	// PMC Warnings St.1
	_CheckFanucPMCActiveAlarmList_St01_Wrn : FB_CheckFanucPMCActiveEvents (
						CheckInterval := T#0S, 
						CurrentPMCActiveAlarmList := _CurrentPMCActiveAlarmListCopy,
						PreviousPMCActiveAlarmList := _PreviousPMCActiveAlarmList,
						StartByte := 410,
						ByteLength := 2,
						SourceId := 101,
						SourceName := 'PMC',
						EventClass := ADR(TC_Events.Wrn01),
						EventDetailer := THIS^
						);
	
	// PMC Warnings St.2
	_CheckFanucPMCActiveAlarmList_St02_Wrn : FB_CheckFanucPMCActiveEvents (
						CheckInterval := T#0S, 
						CurrentPMCActiveAlarmList := _CurrentPMCActiveAlarmListCopy,
						PreviousPMCActiveAlarmList := _PreviousPMCActiveAlarmList,
						StartByte := 412,
						ByteLength := 2,
						SourceId := 102,
						SourceName := 'PMC',
						EventClass := ADR(TC_Events.Wrn02),
						EventDetailer := THIS^
						);
	
	// PMC Warnings St.3
	_CheckFanucPMCActiveAlarmList_St03_Wrn : FB_CheckFanucPMCActiveEvents (
						CheckInterval := T#0S, 
						CurrentPMCActiveAlarmList := _CurrentPMCActiveAlarmListCopy,
						PreviousPMCActiveAlarmList := _PreviousPMCActiveAlarmList,
						StartByte := 414,
						ByteLength := 2,
						SourceId := 103,
						SourceName := 'PMC',
						EventClass := ADR(TC_Events.Wrn03),
						EventDetailer := THIS^
						);
	
	// PMC Warnings St.4
	_CheckFanucPMCActiveAlarmList_St04_Wrn : FB_CheckFanucPMCActiveEvents (
						CheckInterval := T#0S, 
						CurrentPMCActiveAlarmList := _CurrentPMCActiveAlarmListCopy,
						PreviousPMCActiveAlarmList := _PreviousPMCActiveAlarmList,
						StartByte := 416,
						ByteLength := 2,
						SourceId := 104,
						SourceName := 'PMC',
						EventClass := ADR(TC_Events.Wrn04),
						EventDetailer := THIS^
						);
	
	// PMC Warnings St.5
	_CheckFanucPMCActiveAlarmList_St05_Wrn : FB_CheckFanucPMCActiveEvents (
						CheckInterval := T#0S, 
						CurrentPMCActiveAlarmList := _CurrentPMCActiveAlarmListCopy,
						PreviousPMCActiveAlarmList := _PreviousPMCActiveAlarmList,
						StartByte := 418,
						ByteLength := 2,
						SourceId := 105,
						SourceName := 'PMC',
						EventClass := ADR(TC_Events.Wrn05),
						EventDetailer := THIS^
						);
	
	// PMC Warnings St.6
	_CheckFanucPMCActiveAlarmList_St06_Wrn : FB_CheckFanucPMCActiveEvents (
						CheckInterval := T#0S, 
						CurrentPMCActiveAlarmList := _CurrentPMCActiveAlarmListCopy,
						PreviousPMCActiveAlarmList := _PreviousPMCActiveAlarmList,
						StartByte := 420,
						ByteLength := 2,
						SourceId := 106,
						SourceName := 'PMC',
						EventClass := ADR(TC_Events.Wrn06),
						EventDetailer := THIS^
						);
	
	// PMC Warnings St.7
	_CheckFanucPMCActiveAlarmList_St07_Wrn : FB_CheckFanucPMCActiveEvents (
						CheckInterval := T#0S, 
						CurrentPMCActiveAlarmList := _CurrentPMCActiveAlarmListCopy,
						PreviousPMCActiveAlarmList := _PreviousPMCActiveAlarmList,
						StartByte := 422,
						ByteLength := 2,
						SourceId := 107,
						SourceName := 'PMC',
						EventClass := ADR(TC_Events.Wrn07),
						EventDetailer := THIS^
						);
	
	// PMC Warnings St.8
	_CheckFanucPMCActiveAlarmList_St08_Wrn : FB_CheckFanucPMCActiveEvents (
						CheckInterval := T#0S, 
						CurrentPMCActiveAlarmList := _CurrentPMCActiveAlarmListCopy,
						PreviousPMCActiveAlarmList := _PreviousPMCActiveAlarmList,
						StartByte := 424,
						ByteLength := 2,
						SourceId := 108,
						SourceName := 'PMC',
						EventClass := ADR(TC_Events.Wrn08),
						EventDetailer := THIS^
						);
	
	// PMC Warnings St.9
	_CheckFanucPMCActiveAlarmList_St09_Wrn : FB_CheckFanucPMCActiveEvents (
						CheckInterval := T#0S, 
						CurrentPMCActiveAlarmList := _CurrentPMCActiveAlarmListCopy,
						PreviousPMCActiveAlarmList := _PreviousPMCActiveAlarmList,
						StartByte := 426,
						ByteLength := 2,
						SourceId := 109,
						SourceName := 'PMC',
						EventClass := ADR(TC_Events.Wrn09),
						EventDetailer := THIS^
						);
	
	// PMC Warnings St.10
	_CheckFanucPMCActiveAlarmList_St10_Wrn : FB_CheckFanucPMCActiveEvents (
						CheckInterval := T#0S, 
						CurrentPMCActiveAlarmList := _CurrentPMCActiveAlarmListCopy,
						PreviousPMCActiveAlarmList := _PreviousPMCActiveAlarmList,
						StartByte := 428,
						ByteLength := 2,
						SourceId := 110,
						SourceName := 'PMC',
						EventClass := ADR(TC_Events.Wrn10),
						EventDetailer := THIS^
						);
	
	// PMC Warnings St.11
	_CheckFanucPMCActiveAlarmList_St11_Wrn : FB_CheckFanucPMCActiveEvents (
						CheckInterval := T#0S, 
						CurrentPMCActiveAlarmList := _CurrentPMCActiveAlarmListCopy,
						PreviousPMCActiveAlarmList := _PreviousPMCActiveAlarmList,
						StartByte := 430,
						ByteLength := 2,
						SourceId := 111,
						SourceName := 'PMC',
						EventClass := ADR(TC_Events.Wrn11),
						EventDetailer := THIS^
						);
	
	// PMC Warnings St.12
	_CheckFanucPMCActiveAlarmList_St12_Wrn : FB_CheckFanucPMCActiveEvents (
						CheckInterval := T#0S, 
						CurrentPMCActiveAlarmList := _CurrentPMCActiveAlarmListCopy,
						PreviousPMCActiveAlarmList := _PreviousPMCActiveAlarmList,
						StartByte := 432,
						ByteLength := 2,
						SourceId := 112,
						SourceName := 'PMC',
						EventClass := ADR(TC_Events.Wrn12),
						EventDetailer := THIS^
						);
	
	// PMC Warnings St.13
	_CheckFanucPMCActiveAlarmList_St13_Wrn : FB_CheckFanucPMCActiveEvents (
						CheckInterval := T#0S, 
						CurrentPMCActiveAlarmList := _CurrentPMCActiveAlarmListCopy,
						PreviousPMCActiveAlarmList := _PreviousPMCActiveAlarmList,
						StartByte := 434,
						ByteLength := 2,
						SourceId := 113,
						SourceName := 'PMC',
						EventClass := ADR(TC_Events.Wrn13),
						EventDetailer := THIS^
						);
	
//	// PMC Warnings St.14
//	_CheckFanucPMCActiveAlarmList_St14_Wrn : FB_CheckFanucPMCActiveEvents (
//						CheckInterval := T#0S, 
//						CurrentPMCActiveAlarmList := _CurrentPMCActiveAlarmListCopy,
//						PreviousPMCActiveAlarmList := _PreviousPMCActiveAlarmList,
//						StartByte := 436,
//						ByteLength := 2,
//						SourceId := 114,
//						SourceName := 'PMC',
//						EventClass := ADR(TC_Events.Wrn14),
//						EventDetailer := THIS^
//						);
	
//	// PMC Warnings St.15
//	_CheckFanucPMCActiveAlarmList_St15_Wrn : FB_CheckFanucPMCActiveEvents (
//						CheckInterval := T#0S, 
//						CurrentPMCActiveAlarmList := _CurrentPMCActiveAlarmListCopy,
//						PreviousPMCActiveAlarmList := _PreviousPMCActiveAlarmList,
//						StartByte := 438,
//						ByteLength := 2,
//						SourceId := 115,
//						SourceName := 'PMC',
//						EventClass := ADR(TC_Events.Wrn15),
//						EventDetailer := THIS^
//						);
	
//	// PMC Warnings St.16
//	_CheckFanucPMCActiveAlarmList_St16_Wrn : FB_CheckFanucPMCActiveEvents (
//						CheckInterval := T#0S, 
//						CurrentPMCActiveAlarmList := _CurrentPMCActiveAlarmListCopy,
//						PreviousPMCActiveAlarmList := _PreviousPMCActiveAlarmList,
//						StartByte := 440,
//						ByteLength := 2,
//						SourceId := 116,
//						SourceName := 'PMC',
//						EventClass := ADR(TC_Events.Wrn16),
//						EventDetailer := THIS^
//						);
	
//	// PMC Warnings St.17
//	_CheckFanucPMCActiveAlarmList_St17_Wrn : FB_CheckFanucPMCActiveEvents (
//						CheckInterval := T#0S, 
//						CurrentPMCActiveAlarmList := _CurrentPMCActiveAlarmListCopy,
//						PreviousPMCActiveAlarmList := _PreviousPMCActiveAlarmList,
//						StartByte := 442,
//						ByteLength := 2,
//						SourceId := 117,
//						SourceName := 'PMC',
//						EventClass := ADR(TC_Events.Wrn17),
//						EventDetailer := THIS^
//						);
	
//	// PMC Warnings St.18
//	_CheckFanucPMCActiveAlarmList_St18_Wrn : FB_CheckFanucPMCActiveEvents (
//						CheckInterval := T#0S, 
//						CurrentPMCActiveAlarmList := _CurrentPMCActiveAlarmListCopy,
//						PreviousPMCActiveAlarmList := _PreviousPMCActiveAlarmList,
//						StartByte := 444,
//						ByteLength := 2,
//						SourceId := 118,
//						SourceName := 'PMC',
//						EventClass := ADR(TC_Events.Wrn18),
//						EventDetailer := THIS^
//						);
	
//	// PMC Warnings St.19
//	_CheckFanucPMCActiveAlarmList_St19_Wrn : FB_CheckFanucPMCActiveEvents (
//						CheckInterval := T#0S, 
//						CurrentPMCActiveAlarmList := v,
//						PreviousPMCActiveAlarmList := _PreviousPMCActiveAlarmList,
//						StartByte := 446,
//						ByteLength := 2,
//						SourceId := 119,
//						SourceName := 'PMC',
//						EventClass := ADR(TC_Events.Wrn19),
//						EventDetailer := THIS^
//						);
	

						
	// TODO: comment out
	_Gen_Alr  AT %MB600:  ARRAY [0..59] OF BYTE;
	_St00_Alr AT %MB660:  ARRAY [0..39] OF BYTE;
	_St01_Alr AT %MB700:  ARRAY [0..9] OF BYTE;
	_St02_Alr AT %MB710:  ARRAY [0..9] OF BYTE;
	_St03_Alr AT %MB720:  ARRAY [0..9] OF BYTE;
	_St04_Alr AT %MB730:  ARRAY [0..9] OF BYTE;
	_St05_Alr AT %MB740:  ARRAY [0..9] OF BYTE;
	_St06_Alr AT %MB750:  ARRAY [0..9] OF BYTE;
	_St07_Alr AT %MB760:  ARRAY [0..9] OF BYTE;
	_St08_Alr AT %MB770:  ARRAY [0..9] OF BYTE;
	_St09_Alr AT %MB780:  ARRAY [0..9] OF BYTE;
	_St10_Alr AT %MB790:  ARRAY [0..9] OF BYTE;
	_St11_Alr AT %MB800:  ARRAY [0..9] OF BYTE;
	_St12_Alr AT %MB810:  ARRAY [0..9] OF BYTE;
	_St13_Alr AT %MB820:  ARRAY [0..9] OF BYTE;
//	_St14_Alr AT %MB830:  ARRAY [0..9] OF BYTE;
//	_St15_Alr AT %MB840:  ARRAY [0..9] OF BYTE;
//	_St16_Alr AT %MB850:  ARRAY [0..9] OF BYTE;
//	_St17_Alr AT %MB860:  ARRAY [0..9] OF BYTE;
//	_St18_Alr AT %MB870:  ARRAY [0..9] OF BYTE;
//	_St19_Alr AT %MB880:  ARRAY [0..9] OF BYTE;
                         
	_Gen_Wrn  AT %MB1000: ARRAY [0..9] OF BYTE;
	_St01_Wrn AT %MB1010: ARRAY [0..1] OF BYTE;
	_St02_Wrn AT %MB1012: ARRAY [0..1] OF BYTE;
	_St03_Wrn AT %MB1014: ARRAY [0..1] OF BYTE;
	_St04_Wrn AT %MB1016: ARRAY [0..1] OF BYTE;
	_St05_Wrn AT %MB1018: ARRAY [0..1] OF BYTE;
	_St06_Wrn AT %MB1020: ARRAY [0..1] OF BYTE;
	_St07_Wrn AT %MB1022: ARRAY [0..1] OF BYTE;
	_St08_Wrn AT %MB1024: ARRAY [0..1] OF BYTE;
	_St09_Wrn AT %MB1026: ARRAY [0..1] OF BYTE;
	_St10_Wrn AT %MB1028: ARRAY [0..1] OF BYTE;
	_St11_Wrn AT %MB1030: ARRAY [0..1] OF BYTE;
	_St12_Wrn AT %MB1032: ARRAY [0..1] OF BYTE;
	_St13_Wrn AT %MB1034: ARRAY [0..1] OF BYTE;
//	_St14_Wrn AT %MB1036: ARRAY [0..1] OF BYTE;
//	_St15_Wrn AT %MB1038: ARRAY [0..1] OF BYTE;
//	_St16_Wrn AT %MB1040: ARRAY [0..1] OF BYTE;
//	_St17_Wrn AT %MB1042: ARRAY [0..1] OF BYTE;
//	_St18_Wrn AT %MB1044: ARRAY [0..1] OF BYTE;
//	_St19_Wrn AT %MB1046: ARRAY [0..1] OF BYTE;

END_VAR

_CheckTimer();

IF Enabled  AND (_CheckInterval > T#0MS) THEN
	IF _CheckTimer.Q THEN
		// Freeze current list into local copy to avoid concurrency problems with ADS
		MEMCPY(ADR(_CurrentPMCActiveAlarmListCopy), ADR(_CurrentPMCActiveAlarmList), NUM_PMC_EVENTS / 8);
		// Update all
		UpdateActiveEventList();
		_CheckTimer.IN := FALSE;
	ELSE
		_CheckTimer.IN := TRUE;
	END_IF
ELSE
	_CheckTimer.IN := FALSE;
END_IF


// Alarms (cyclic call)
_CheckFanucPMCActiveAlarmList_Gen_Alr();
_CheckFanucPMCActiveAlarmList_St00_Alr();
_CheckFanucPMCActiveAlarmList_St01_Alr();
_CheckFanucPMCActiveAlarmList_St02_Alr();
_CheckFanucPMCActiveAlarmList_St03_Alr();
_CheckFanucPMCActiveAlarmList_St04_Alr();
_CheckFanucPMCActiveAlarmList_St05_Alr();
_CheckFanucPMCActiveAlarmList_St06_Alr();
_CheckFanucPMCActiveAlarmList_St07_Alr();
_CheckFanucPMCActiveAlarmList_St08_Alr();
_CheckFanucPMCActiveAlarmList_St09_Alr();
_CheckFanucPMCActiveAlarmList_St10_Alr();
_CheckFanucPMCActiveAlarmList_St11_Alr();
_CheckFanucPMCActiveAlarmList_St12_Alr();
_CheckFanucPMCActiveAlarmList_St13_Alr();
//_CheckFanucPMCActiveAlarmList_St14_Alr();
//_CheckFanucPMCActiveAlarmList_St15_Alr();
//_CheckFanucPMCActiveAlarmList_St16_Alr();
//_CheckFanucPMCActiveAlarmList_St17_Alr();
//_CheckFanucPMCActiveAlarmList_St18_Alr();
//_CheckFanucPMCActiveAlarmList_St19_Alr();

// Warnings (cyclic call)
_CheckFanucPMCActiveAlarmList_Gen_Wrn();
_CheckFanucPMCActiveAlarmList_St01_Wrn();
_CheckFanucPMCActiveAlarmList_St02_Wrn();
_CheckFanucPMCActiveAlarmList_St03_Wrn();
_CheckFanucPMCActiveAlarmList_St04_Wrn();
_CheckFanucPMCActiveAlarmList_St05_Wrn();
_CheckFanucPMCActiveAlarmList_St06_Wrn();
_CheckFanucPMCActiveAlarmList_St07_Wrn();
_CheckFanucPMCActiveAlarmList_St08_Wrn();
_CheckFanucPMCActiveAlarmList_St09_Wrn();
_CheckFanucPMCActiveAlarmList_St10_Wrn();
_CheckFanucPMCActiveAlarmList_St11_Wrn();
_CheckFanucPMCActiveAlarmList_St12_Wrn();
_CheckFanucPMCActiveAlarmList_St13_Wrn();
//_CheckFanucPMCActiveAlarmList_St14_Wrn();
//_CheckFanucPMCActiveAlarmList_St15_Wrn();
//_CheckFanucPMCActiveAlarmList_St16_Wrn();
//_CheckFanucPMCActiveAlarmList_St17_Wrn();
//_CheckFanucPMCActiveAlarmList_St18_Wrn();
//_CheckFanucPMCActiveAlarmList_St19_Wrn();

PROPERTY PUBLIC CheckInterval : TIME
GET
CheckInterval := _CheckInterval;
END_GET
SET
_CheckTimer.PT := _CheckInterval;

//// Alarms
//_CheckFanucPMCActiveAlarmList_Gen_Alr.CheckInterval := _CheckInterval;
//_CheckFanucPMCActiveAlarmList_St00_Alr.CheckInterval := _CheckInterval;
//_CheckFanucPMCActiveAlarmList_St01_Alr.CheckInterval := _CheckInterval;
//_CheckFanucPMCActiveAlarmList_St02_Alr.CheckInterval := _CheckInterval;
//_CheckFanucPMCActiveAlarmList_St03_Alr.CheckInterval := _CheckInterval;
//_CheckFanucPMCActiveAlarmList_St04_Alr.CheckInterval := _CheckInterval;
//_CheckFanucPMCActiveAlarmList_St05_Alr.CheckInterval := _CheckInterval;
//_CheckFanucPMCActiveAlarmList_St06_Alr.CheckInterval := _CheckInterval;
//_CheckFanucPMCActiveAlarmList_St07_Alr.CheckInterval := _CheckInterval;
//_CheckFanucPMCActiveAlarmList_St08_Alr.CheckInterval := _CheckInterval;
//_CheckFanucPMCActiveAlarmList_St09_Alr.CheckInterval := _CheckInterval;
//_CheckFanucPMCActiveAlarmList_St10_Alr.CheckInterval := _CheckInterval;
//_CheckFanucPMCActiveAlarmList_St11_Alr.CheckInterval := _CheckInterval;
//_CheckFanucPMCActiveAlarmList_St12_Alr.CheckInterval := _CheckInterval;
//_CheckFanucPMCActiveAlarmList_St13_Alr.CheckInterval := _CheckInterval;
//_CheckFanucPMCActiveAlarmList_St14_Alr.CheckInterval := _CheckInterval;
//_CheckFanucPMCActiveAlarmList_St15_Alr.CheckInterval := _CheckInterval;
//_CheckFanucPMCActiveAlarmList_St16_Alr.CheckInterval := _CheckInterval;
////_CheckFanucPMCActiveAlarmList_St17_Alr.CheckInterval := _CheckInterval;
////_CheckFanucPMCActiveAlarmList_St18_Alr.CheckInterval := _CheckInterval;
////_CheckFanucPMCActiveAlarmList_St19_Alr.CheckInterval := _CheckInterval;

//// Warnings
//_CheckFanucPMCActiveAlarmList_Gen_Wrn.CheckInterval := _CheckInterval;
//_CheckFanucPMCActiveAlarmList_St01_Wrn.CheckInterval := _CheckInterval;
//_CheckFanucPMCActiveAlarmList_St02_Wrn.CheckInterval := _CheckInterval;
//_CheckFanucPMCActiveAlarmList_St03_Wrn.CheckInterval := _CheckInterval;
//_CheckFanucPMCActiveAlarmList_St04_Wrn.CheckInterval := _CheckInterval;
//_CheckFanucPMCActiveAlarmList_St05_Wrn.CheckInterval := _CheckInterval;
//_CheckFanucPMCActiveAlarmList_St06_Wrn.CheckInterval := _CheckInterval;
//_CheckFanucPMCActiveAlarmList_St07_Wrn.CheckInterval := _CheckInterval;
//_CheckFanucPMCActiveAlarmList_St08_Wrn.CheckInterval := _CheckInterval;
//_CheckFanucPMCActiveAlarmList_St09_Wrn.CheckInterval := _CheckInterval;
//_CheckFanucPMCActiveAlarmList_St10_Wrn.CheckInterval := _CheckInterval;
//_CheckFanucPMCActiveAlarmList_St11_Wrn.CheckInterval := _CheckInterval;
//_CheckFanucPMCActiveAlarmList_St12_Wrn.CheckInterval := _CheckInterval;
//_CheckFanucPMCActiveAlarmList_St13_Wrn.CheckInterval := _CheckInterval;
//_CheckFanucPMCActiveAlarmList_St14_Wrn.CheckInterval := _CheckInterval;
//_CheckFanucPMCActiveAlarmList_St15_Wrn.CheckInterval := _CheckInterval;
//_CheckFanucPMCActiveAlarmList_St16_Wrn.CheckInterval := _CheckInterval;
////_CheckFanucPMCActiveAlarmList_St17_Wrn.CheckInterval := _CheckInterval;
////_CheckFanucPMCActiveAlarmList_St18_Wrn.CheckInterval := _CheckInterval;
////_CheckFanucPMCActiveAlarmList_St19_Wrn.CheckInterval := _CheckInterval;
END_SET
END_PROPERTY

METHOD PUBLIC ClearAll : BOOL
VAR
	_TcEventFilter : FB_TcEventFilter;
END_VAR
// Alarms
_CheckFanucPMCActiveAlarmList_St01_Alr.ClearAll();
_CheckFanucPMCActiveAlarmList_St02_Alr.ClearAll();
_CheckFanucPMCActiveAlarmList_St03_Alr.ClearAll();
_CheckFanucPMCActiveAlarmList_St04_Alr.ClearAll();
_CheckFanucPMCActiveAlarmList_St05_Alr.ClearAll();
_CheckFanucPMCActiveAlarmList_St06_Alr.ClearAll();
_CheckFanucPMCActiveAlarmList_St07_Alr.ClearAll();
_CheckFanucPMCActiveAlarmList_St08_Alr.ClearAll();
_CheckFanucPMCActiveAlarmList_St09_Alr.ClearAll();
_CheckFanucPMCActiveAlarmList_St10_Alr.ClearAll();
_CheckFanucPMCActiveAlarmList_St11_Alr.ClearAll();
_CheckFanucPMCActiveAlarmList_St12_Alr.ClearAll();
_CheckFanucPMCActiveAlarmList_St13_Alr.ClearAll();
//_CheckFanucPMCActiveAlarmList_St14_Alr.ClearAll();
//_CheckFanucPMCActiveAlarmList_St15_Alr.ClearAll();
//_CheckFanucPMCActiveAlarmList_St16_Alr.ClearAll();
//_CheckFanucPMCActiveAlarmList_St17_Alr.ClearAll();
//_CheckFanucPMCActiveAlarmList_St18_Alr.ClearAll();
//_CheckFanucPMCActiveAlarmList_St19_Alr.ClearAll();

// Warnings
_CheckFanucPMCActiveAlarmList_St01_Wrn.ClearAll();
_CheckFanucPMCActiveAlarmList_St02_Wrn.ClearAll();
_CheckFanucPMCActiveAlarmList_St03_Wrn.ClearAll();
_CheckFanucPMCActiveAlarmList_St04_Wrn.ClearAll();
_CheckFanucPMCActiveAlarmList_St05_Wrn.ClearAll();
_CheckFanucPMCActiveAlarmList_St06_Wrn.ClearAll();
_CheckFanucPMCActiveAlarmList_St07_Wrn.ClearAll();
_CheckFanucPMCActiveAlarmList_St08_Wrn.ClearAll();
_CheckFanucPMCActiveAlarmList_St09_Wrn.ClearAll();
_CheckFanucPMCActiveAlarmList_St10_Wrn.ClearAll();
_CheckFanucPMCActiveAlarmList_St11_Wrn.ClearAll();
_CheckFanucPMCActiveAlarmList_St12_Wrn.ClearAll();
_CheckFanucPMCActiveAlarmList_St13_Wrn.ClearAll();
//_CheckFanucPMCActiveAlarmList_St14_Wrn.ClearAll();
//_CheckFanucPMCActiveAlarmList_St15_Wrn.ClearAll();
//_CheckFanucPMCActiveAlarmList_St16_Wrn.ClearAll();
//_CheckFanucPMCActiveAlarmList_St17_Wrn.ClearAll();
//_CheckFanucPMCActiveAlarmList_St18_Wrn.ClearAll();
//_CheckFanucPMCActiveAlarmList_St19_Wrn.ClearAll();
END_METHOD

PROPERTY PUBLIC Enabled : BOOL
GET
Enabled := _Enabled;
END_GET
SET
_Enabled := Enabled;

// Alarms
_CheckFanucPMCActiveAlarmList_Gen_Alr.Enabled := _Enabled;
_CheckFanucPMCActiveAlarmList_St00_Alr.Enabled := _Enabled;
_CheckFanucPMCActiveAlarmList_St01_Alr.Enabled := _Enabled;
_CheckFanucPMCActiveAlarmList_St02_Alr.Enabled := _Enabled;
_CheckFanucPMCActiveAlarmList_St03_Alr.Enabled := _Enabled;
_CheckFanucPMCActiveAlarmList_St04_Alr.Enabled := _Enabled;
_CheckFanucPMCActiveAlarmList_St05_Alr.Enabled := _Enabled;
_CheckFanucPMCActiveAlarmList_St06_Alr.Enabled := _Enabled;
_CheckFanucPMCActiveAlarmList_St07_Alr.Enabled := _Enabled;
_CheckFanucPMCActiveAlarmList_St08_Alr.Enabled := _Enabled;
_CheckFanucPMCActiveAlarmList_St09_Alr.Enabled := _Enabled;
_CheckFanucPMCActiveAlarmList_St10_Alr.Enabled := _Enabled;
_CheckFanucPMCActiveAlarmList_St11_Alr.Enabled := _Enabled;
_CheckFanucPMCActiveAlarmList_St12_Alr.Enabled := _Enabled;
_CheckFanucPMCActiveAlarmList_St13_Alr.Enabled := _Enabled;
//_CheckFanucPMCActiveAlarmList_St14_Alr.Enabled := _Enabled;
//_CheckFanucPMCActiveAlarmList_St15_Alr.Enabled := _Enabled;
//_CheckFanucPMCActiveAlarmList_St16_Alr.Enabled := _Enabled;
//_CheckFanucPMCActiveAlarmList_St17_Alr.Enabled := _Enabled;
//_CheckFanucPMCActiveAlarmList_St18_Alr.Enabled := _Enabled;
//_CheckFanucPMCActiveAlarmList_St19_Alr.Enabled := _Enabled;

// Warnings
_CheckFanucPMCActiveAlarmList_Gen_Wrn.Enabled := _Enabled;
_CheckFanucPMCActiveAlarmList_St01_Wrn.Enabled := _Enabled;
_CheckFanucPMCActiveAlarmList_St02_Wrn.Enabled := _Enabled;
_CheckFanucPMCActiveAlarmList_St03_Wrn.Enabled := _Enabled;
_CheckFanucPMCActiveAlarmList_St04_Wrn.Enabled := _Enabled;
_CheckFanucPMCActiveAlarmList_St05_Wrn.Enabled := _Enabled;
_CheckFanucPMCActiveAlarmList_St06_Wrn.Enabled := _Enabled;
_CheckFanucPMCActiveAlarmList_St07_Wrn.Enabled := _Enabled;
_CheckFanucPMCActiveAlarmList_St08_Wrn.Enabled := _Enabled;
_CheckFanucPMCActiveAlarmList_St09_Wrn.Enabled := _Enabled;
_CheckFanucPMCActiveAlarmList_St10_Wrn.Enabled := _Enabled;
_CheckFanucPMCActiveAlarmList_St11_Wrn.Enabled := _Enabled;
_CheckFanucPMCActiveAlarmList_St12_Wrn.Enabled := _Enabled;
_CheckFanucPMCActiveAlarmList_St13_Wrn.Enabled := _Enabled;
//_CheckFanucPMCActiveAlarmList_St14_Wrn.Enabled := _Enabled;
//_CheckFanucPMCActiveAlarmList_St15_Wrn.Enabled := _Enabled;
//_CheckFanucPMCActiveAlarmList_St16_Wrn.Enabled := _Enabled;
//_CheckFanucPMCActiveAlarmList_St17_Wrn.Enabled := _Enabled;
//_CheckFanucPMCActiveAlarmList_St18_Wrn.Enabled := _Enabled;
//_CheckFanucPMCActiveAlarmList_St19_Wrn.Enabled := _Enabled;
END_SET
END_PROPERTY

METHOD FB_init : BOOL
VAR_INPUT
	bInitRetains : BOOL; // if TRUE, the retain variables are initialized (warm start / cold start)
	bInCopyCode : BOOL;  // if TRUE, the instance afterwards gets moved into the copy code (online change)
	CheckInterval : TIME;
	CurrentPMCActiveAlarmList : REFERENCE TO ARRAY [0..NUM_PMC_EVENTS / 8 - 1] OF BYTE;
END_VAR
_CheckInterval := CheckInterval;
_CheckTimer.PT := _CheckInterval;

IF __ISVALIDREF(CurrentPMCActiveAlarmList) THEN
	_CurrentPMCActiveAlarmList REF= CurrentPMCActiveAlarmList;
END_IF
END_METHOD

METHOD GetDetail : STRING(255)
VAR_INPUT
	TcAlarm	: REFERENCE TO Tc3_EventLogger.FB_TcAlarm;
END_VAR
VAR
	_Detail : STRING(255);
END_VAR
_Detail := '';

// St.01 Alarms
IF TcAlarm.EqualsToEventClass(TC_EVENT_CLASSES.Alr01) THEN
	CASE TcAlarm.nEventId OF
		0: _Detail := 'This is alarm 0 of St.1';
		1: _Detail := 'This is alarm 1 of St.1';
		2: _Detail := 'This is alarm 2 of St.1';
		3: _Detail := 'This is alarm 3 of St.1';
		//4: _Detail := Main._CurrentUser.Name;
		//5: _Detail := GlobalUser.GlobalUser.Name;
	END_CASE
END_IF

// St.01 Warnings
IF TcAlarm.EqualsToEventClass(TC_EVENT_CLASSES.Wrn01) THEN
	CASE TcAlarm.nEventId OF
		0: _Detail := 'This is warning 0 of St.1';
		1: _Detail := 'This is warning 1 of St.1';
		2: _Detail := 'This is warning 2 of St.1';
		3: _Detail := 'This is warning 3 of St.1';
	END_CASE
END_IF

GetDetail := _Detail;
END_METHOD

METHOD PUBLIC ReSync : BOOL
// Force resynchronization of active events
//		- Clear all raised events
//		- Reset previous memory buffer
//		- Update active event list
ClearAll();
MemSet(ADR(_PreviousPMCActiveAlarmList), 0, SIZEOF(_PreviousPMCActiveAlarmList));
UpdateActiveEventList();
END_METHOD

METHOD PUBLIC UpdateActiveEventList : BOOL
// Alarms
_CheckFanucPMCActiveAlarmList_Gen_Alr.UpdateActiveEventList();
_CheckFanucPMCActiveAlarmList_St00_Alr.UpdateActiveEventList();
_CheckFanucPMCActiveAlarmList_St01_Alr.UpdateActiveEventList();
_CheckFanucPMCActiveAlarmList_St02_Alr.UpdateActiveEventList();
_CheckFanucPMCActiveAlarmList_St03_Alr.UpdateActiveEventList();
_CheckFanucPMCActiveAlarmList_St04_Alr.UpdateActiveEventList();
_CheckFanucPMCActiveAlarmList_St05_Alr.UpdateActiveEventList();
_CheckFanucPMCActiveAlarmList_St06_Alr.UpdateActiveEventList();
_CheckFanucPMCActiveAlarmList_St07_Alr.UpdateActiveEventList();
_CheckFanucPMCActiveAlarmList_St08_Alr.UpdateActiveEventList();
_CheckFanucPMCActiveAlarmList_St09_Alr.UpdateActiveEventList();
_CheckFanucPMCActiveAlarmList_St10_Alr.UpdateActiveEventList();
_CheckFanucPMCActiveAlarmList_St11_Alr.UpdateActiveEventList();
_CheckFanucPMCActiveAlarmList_St12_Alr.UpdateActiveEventList();
_CheckFanucPMCActiveAlarmList_St13_Alr.UpdateActiveEventList();
//_CheckFanucPMCActiveAlarmList_St14_Alr.UpdateActiveEventList();
//_CheckFanucPMCActiveAlarmList_St15_Alr.UpdateActiveEventList();
//_CheckFanucPMCActiveAlarmList_St16_Alr.UpdateActiveEventList();
//_CheckFanucPMCActiveAlarmList_St17_Alr.UpdateActiveEventList();
//_CheckFanucPMCActiveAlarmList_St18_Alr.UpdateActiveEventList();
//_CheckFanucPMCActiveAlarmList_St19_Alr.UpdateActiveEventList();

// Warnings
_CheckFanucPMCActiveAlarmList_Gen_Wrn.UpdateActiveEventList();
_CheckFanucPMCActiveAlarmList_St01_Wrn.UpdateActiveEventList();
_CheckFanucPMCActiveAlarmList_St02_Wrn.UpdateActiveEventList();
_CheckFanucPMCActiveAlarmList_St03_Wrn.UpdateActiveEventList();
_CheckFanucPMCActiveAlarmList_St04_Wrn.UpdateActiveEventList();
_CheckFanucPMCActiveAlarmList_St05_Wrn.UpdateActiveEventList();
_CheckFanucPMCActiveAlarmList_St06_Wrn.UpdateActiveEventList();
_CheckFanucPMCActiveAlarmList_St07_Wrn.UpdateActiveEventList();
_CheckFanucPMCActiveAlarmList_St08_Wrn.UpdateActiveEventList();
_CheckFanucPMCActiveAlarmList_St09_Wrn.UpdateActiveEventList();
_CheckFanucPMCActiveAlarmList_St10_Wrn.UpdateActiveEventList();
_CheckFanucPMCActiveAlarmList_St11_Wrn.UpdateActiveEventList();
_CheckFanucPMCActiveAlarmList_St12_Wrn.UpdateActiveEventList();
_CheckFanucPMCActiveAlarmList_St13_Wrn.UpdateActiveEventList();
//_CheckFanucPMCActiveAlarmList_St14_Wrn.UpdateActiveEventList();
//_CheckFanucPMCActiveAlarmList_St15_Wrn.UpdateActiveEventList();
//_CheckFanucPMCActiveAlarmList_St16_Wrn.UpdateActiveEventList();
//_CheckFanucPMCActiveAlarmList_St17_Wrn.UpdateActiveEventList();
//_CheckFanucPMCActiveAlarmList_St18_Wrn.UpdateActiveEventList();
//_CheckFanucPMCActiveAlarmList_St19_Wrn.UpdateActiveEventList();
END_METHOD

END_FUNCTION_BLOCK

// ---- FBs/Events/FB_CheckFanucPMCActiveEvents.TcPOU
FUNCTION_BLOCK FB_CheckFanucPMCActiveEvents
VAR_INPUT
	Enabled : BOOL;
END_VAR
VAR

	{attribute 'hide'}
	_PMCEvents : ARRAY[0..NUM_PMC_EVENTS] OF FB_TcAlarm;

	{attribute 'hide'}
	_CurrentPMCActiveAlarmList : REFERENCE TO ARRAY [0..NUM_PMC_EVENTS / 8 - 1] OF BYTE;

	{attribute 'hide'}
	_PreviousPMCActiveAlarmList : REFERENCE TO ARRAY [0..NUM_PMC_EVENTS / 8 - 1] OF BYTE;
	
	{attribute 'hide'}
	_TcEventLogger : FB_TcEventLogger;	

	{attribute 'hide'}
	_TcSourceInfo : FB_TcSourceInfo;

	{attribute 'hide'}
	_CheckInterval : TIME;
	
	{attribute 'hide'}
	_CheckTimer : TON;
	
	{attribute 'hide'}
	_StartByte : UDINT := 0;

	{attribute 'hide'}
	_ByteLength : UDINT := 0;

	{attribute 'hide'}
	_EventClass : POINTER TO TcEventEntry;
	
	{attribute 'hide'}
	_EventDetailer : I_EventDetailer;
	
END_VAR

_CheckTimer();

IF Enabled  AND (_CheckInterval > T#0MS) THEN
	IF _CheckTimer.Q THEN
		THIS^.UpdateActiveEventList();
		_CheckTimer.IN := FALSE;
	ELSE
		_CheckTimer.IN := TRUE;
	END_IF
ELSE
	_CheckTimer.IN := FALSE;
END_IF

METHOD PRIVATE BinarySearch : BOOL
VAR_INPUT
	FirstByteIndex : UDINT;
	LastByteIndex : UDINT;
END_VAR
VAR 
	_i : UDINT;
	_StateChanged : INT;
	_EventIndex : UDINT;
	_pTcEventEntry : POINTER TO TcEventEntry;
	_MiddleByteIndex : UDINT;
	_TcAlarm : FB_TcAlarm;
	_refTcAlarm : REFERENCE TO FB_TcAlarm REF= _TcAlarm;
	_hr : HRESULT;
END_VAR
IF FirstByteIndex = LastByteIndex THEN
	IF _PreviousPMCActiveAlarmList[FirstByteIndex] <> _CurrentPMCActiveAlarmList[FirstByteIndex] THEN
		// Check every bit for change: (X = 2^BitPos)
		// | Current | Previous | Current - Previous | StateChanged
		// |    0     |    0    |         0          | No change
		// |    0     |    1    |      -X < 0        | Event gone
		// |    1     |    0    |       X > 0        | Event coming
		// |    1     |    1    |         0          | No change
		_pTcEventEntry := _EventClass;
		FOR _i := 0 TO 7 DO
			_StateChanged := BYTE_TO_INT(_CurrentPMCActiveAlarmList[FirstByteIndex] AND SHL(16#1, _i)) - BYTE_TO_INT(_PreviousPMCActiveAlarmList[FirstByteIndex] AND SHL(16#1, _i));
			IF _StateChanged < 0 THEN
				// Event gone
				_EventIndex := (FirstByteIndex - _StartByte) * 8 + _i;
				// Clear event
				IF _PMCEvents[_EventIndex].bRaised THEN
					_PMCEvents[_EventIndex].Clear(0, TRUE);
				END_IF
			END_IF
			IF _StateChanged > 0 THEN
				// Event coming
				_EventIndex := (FirstByteIndex - _StartByte) * 8 + _i;
				// Create event instance if not already created
				IF _PMCEvents[_EventIndex].nUniqueId = 0 THEN
					_PMCEvents[_EventIndex].CreateEx(_pTcEventEntry[_EventIndex], FALSE, GetSourceInfo());
				END_IF
				// Raise event (if not already raised)
				IF NOT _PMCEvents[_EventIndex].bRaised THEN
					SetParameters(_PMCEvents[_EventIndex]);
					_PMCEvents[_EventIndex].Raise(0);
				END_IF
			END_IF		
		END_FOR		
	END_IF
ELSE
	_MiddleByteIndex := FirstByteIndex + LREAL_TO_UDINT(FLOOR((LastByteIndex - FirstByteIndex) / 2));
	// Check first half (recursive)
	IF MEMCMP(ADR(_PreviousPMCActiveAlarmList[FirstByteIndex]), ADR(_CurrentPMCActiveAlarmList[FirstByteIndex]), (_MiddleByteIndex + 1 - FirstByteIndex)) <> 0 THEN
		THIS^.BinarySearch(FirstByteIndex, _MiddleByteIndex);
	END_IF
	// Check second half (recursive)
	IF MEMCMP(ADR(_PreviousPMCActiveAlarmList[_MiddleByteIndex + 1]), ADR(_CurrentPMCActiveAlarmList[_MiddleByteIndex + 1]), (LastByteIndex - _MiddleByteIndex)) <> 0 THEN
		THIS^.BinarySearch(_MiddleByteIndex + 1, LastByteIndex);
	END_IF
END_IF
END_METHOD

PROPERTY PUBLIC ByteLength : UDINT
GET
ByteLength := _ByteLength;
END_GET
END_PROPERTY

PROPERTY PUBLIC CheckInterval : TIME
GET
CheckInterval := _CheckInterval;
END_GET
SET
_CheckInterval := CheckInterval;
_CheckTimer.PT := _CheckInterval;
END_SET
END_PROPERTY

METHOD PUBLIC ClearAll : BOOL
VAR
	_TcEventFilter : FB_TcEventFilter;
END_VAR
//_TcEventFilter.Clear().EventClass.EqualTo(_EventClass);
//_TcEventLogger.ClearAlarms(0, FALSE, _TcEventFilter);
END_METHOD

METHOD FB_init : BOOL
VAR_INPUT
	bInitRetains : BOOL; // if TRUE, the retain variables are initialized (warm start / cold start)
	bInCopyCode : BOOL;  // if TRUE, the instance afterwards gets moved into the copy code (online change)
	CheckInterval : TIME;
	CurrentPMCActiveAlarmList : REFERENCE TO ARRAY [0..NUM_PMC_EVENTS / 8 - 1] OF BYTE;
	PreviousPMCActiveAlarmList : REFERENCE TO ARRAY [0..NUM_PMC_EVENTS / 8 - 1] OF BYTE;
	StartByte : UDINT;
	ByteLength : UDINT;
	SourceId : UDINT := 0;
	SourceName : STRING[80] := '';
	EventClass : POINTER TO TcEventEntry;
	EventDetailer : I_EventDetailer;
END_VAR
_CheckInterval := CheckInterval;
_CheckTimer.PT := _CheckInterval;

_StartByte := StartByte;
_ByteLength := ByteLength;

_EventClass := EventClass;

InitSource(SourceId, SourceName);

IF __ISVALIDREF(CurrentPMCActiveAlarmList) THEN
	_CurrentPMCActiveAlarmList REF= CurrentPMCActiveAlarmList;
END_IF

IF __ISVALIDREF(PreviousPMCActiveAlarmList) THEN
	_PreviousPMCActiveAlarmList REF= PreviousPMCActiveAlarmList;
END_IF

_EventDetailer := EventDetailer;
END_METHOD

METHOD PRIVATE GetSourceInfo : I_TcSourceInfo
GetSourceInfo := _TcSourceInfo;
END_METHOD

METHOD PRIVATE InitSource : BOOL
VAR_INPUT
	Id : UDINT;
	Name : STRING(80);
END_VAR
_TcSourceInfo.Clear();
_TcSourceInfo.nId := ID;
_TcSourceInfo.sName := Name;
END_METHOD

METHOD PRIVATE SetParameters : BOOL
VAR_INPUT
	TcAlarm : REFERENCE TO FB_TcAlarm;
END_VAR
VAR
	_Detail : STRING(512);
END_VAR
IF _EventDetailer <> 0 THEN
	_Detail := _EventDetailer.GetDetail(TcAlarm);
END_IF

TcAlarm.ipArguments.Clear();

IF LEn(_Detail) <> 0 THEN
	TcAlarm.ipArguments.AddString(_Detail);
END_IF
END_METHOD

PROPERTY PUBLIC SourceId : UDINT
GET
SourceId := _TcSourceInfo.nId;
END_GET
END_PROPERTY

PROPERTY PUBLIC SourceName : STRING(80)
GET
SourceName := _TcSourceInfo.sName;
END_GET
END_PROPERTY

PROPERTY PUBLIC StartByte : UDINT
GET
StartByte := _StartByte;
END_GET
END_PROPERTY

METHOD PUBLIC UpdateActiveEventList : BOOL
VAR
	_i : UINT;
	_j : UINT;
	_Found : BOOL;	
	_TcAlarm : FB_TcAlarm;
	_refTcAlarm : REFERENCE TO FB_TcAlarm REF= _TcAlarm;
	_iTcSourceInfo : I_TcSourceInfo;
	_hr : HRESULT;
END_VAR
IF SIZEOF(_PreviousPMCActiveAlarmList) <> SIZEOF(_CurrentPMCActiveAlarmList) THEN
	UpdateActiveEventList := FALSE;
	RETURN;
END_IF

IF MEMCMP(ADR(_PreviousPMCActiveAlarmList) + _StartByte, ADR(_CurrentPMCActiveAlarmList) + _StartByte, _ByteLength) <> 0 THEN
	
	// Explore alarms and manage going and coming
	IF SIZEOF(_CurrentPMCActiveAlarmList) > 0 THEN
		BinarySearch(_StartByte, _StartByte + _ByteLength - 1);
	END_IF
	
	// Update previous list with current list
	MEMCPY(ADR(_PreviousPMCActiveAlarmList) + _StartByte, ADR(_CurrentPMCActiveAlarmList) + _StartByte, _ByteLength);

END_IF

UpdateActiveEventList := TRUE;
END_METHOD

END_FUNCTION_BLOCK

// ---- FBs/Database/PRG_MSSQL_spCMD_AbortProduction.TcPOU
PROGRAM PRG_MSSQL_spCMD_AbortProduction
VAR_INPUT
	Execute					: BOOL;
	Enable					: BOOL;
END_VAR
VAR_OUTPUT
	Error					: BOOL;
	ErrorID					: DINT;
	Done					: BOOL;
	Busy					: BOOL;
	tcMessage 				: I_TcMessage;
	Q_tElapsedTime			: TIME;
END_VAR
VAR
	RTRIG_Execute			: R_TRIG;
	iState					: INT := -1;
	return_value				: DINT;
END_VAR
VAR_IN_OUT
	fbSQLResult				: FB_SQLResultEvt;
	fbSQLStoredProcedure	: FB_SQLStoredProcedureEvt;
END_VAR

RTRIG_Execute(CLK := Execute AND Enable);
IF(RTRIG_Execute.Q) THEN
	 Done							:= FALSE;
	 Error							:= FALSE;
	 ErrorID						:= 0;
	 
	 iState							:= 0;
ELSIF NOT Execute AND NOT Busy THEN
	Busy			:= FALSE;
	Done			:= FALSE;
	Error			:= FALSE;
	
	iState := -1;
END_IF
 
 CASE iState OF
 
	 0:
		Busy								:= TRUE;
		iState 								:= 10;
		
	10:
		IF fbSQLStoredProcedure.ExecuteDataReturn(pParameterStrc := ADR(return_value), cbParameterStrc := SIZEOF(return_value), pSQLDBResult := ADR(fbSqlResult)) THEN
			IF fbSQLStoredProcedure.bError THEN
				tcMessage := fbSQLStoredProcedure.ipTcResult;
				
				iState 							:= 1010;
			ELSE
				iState 							:= 20;
			END_IF    
		END_IF
		
	20:
		IF return_value = 0 THEN
			iState 								:= 999;	
		ELSE
			iState 								:= 1020;	
		END_IF
		
	999:
		Done			:= TRUE;
		Busy			:= FALSE;
		
 END_CASE 
 
IF iState > 1000 THEN
	Error 		:= TRUE;
	ErrorID	 	:= iState;
	Busy	 	:= FALSE;
	iState := -1;
END_IF

END_PROGRAM

// ---- FCs/FC_BYTE_TO_BOOLARR.TcPOU
FUNCTION FC_BYTE_TO_BOOLARR
VAR_INPUT
	pMyBool : POINTER TO BOOL; // Destination 
	pMyByte : POINTER TO BYTE; // Source   
	nSize	: UINT;               
END_VAR
VAR
    i : UINT;                       
	myBools : ARRAY[0..7] OF BOOL; 
END_VAR

FOR i:= 0 TO nSize-1 BY 8 DO
	myBools := FC_BYTE_TO_BOOLBYTE(pMyByte[i/8]);
	MEMCPY(ADR(pMyBool[i]), ADR(myBools), SIZEOF(myBools));
END_FOR

END_FUNCTION

// ---- FCs/FC_BYTE_TO_BOOLBYTE.TcPOU
FUNCTION FC_BYTE_TO_BOOLBYTE : ARRAY[0..7] OF BOOL
VAR_INPUT
	myByte : REFERENCE TO BYTE;
END_VAR
VAR
    i : USINT;
END_VAR

FOR i := 0 TO 7 DO
    FC_BYTE_TO_BOOLBYTE[i] := (myByte AND (SHL(1,i))) <> 0;
END_FOR

END_FUNCTION

// ---- POUs/MAIN_SERVICE.TcPOU
PROGRAM MAIN_SERVICE
VAR
	
// HMI - Tools	
	NT_CNCScreenDisplay: NT_StartProcess;
	NT_ProgramTransferTool: NT_StartProcess;
	NT_TaskManager: NT_StartProcess;
	NT_OnScreenKeyboard: NT_StartProcess;
	NT_CloseBrowser: NT_StartProcess;
	NT_FanucLadder: NT_StartProcess;
	NT_FlyCad: NT_StartProcess;
	NT_OpenExe : NT_StartProcess;
	NT_CloseExe : NT_StartProcess;
	
	TON_OpenPage : TON;
	
	GetTime								: FB_LocalSystemTime := ( bEnable := TRUE, dwCycle := 1 );	
	
	otTON						: OTSTRUCT;
	otTOFF						: OTSTRUCT;
	otTDOWN						: OTSTRUCT;
	otTTotal					: OTSTRUCT;
	TempSum						: REAL;
	TempTime1					: REAL;
	TempTime2					: REAL;
	TempTime3					: REAL;
	RTON_ON					: FB_RetainTimer;
	RTON_OFF				: FB_RetainTimer;
	RTON_DOWN				: FB_RetainTimer;

	fbGetCurTaskIndex : GETCURTASKINDEX;
	
	TON_OvrMultFeedback : TON;
	OvrMultiplierOld	: USINT;
	_iDataPos : INT;
	i : INT;
	RTRIG_ClearAlarm	: R_TRIG;
	TcSourceInfo	: FB_TcSourceInfo;
	fbRefresh : FB_Refresh;
	MSSQL_Events					: DUT_Events;
	Marker_Events					: DUT_Events;
	DataRequest_Events				: DUT_Events;
	
	TON_DelayMarkerConnected	: TON;
	fbDoublingTriggerGood : FB_DoublingTrigger;
	fbDoublingTriggerBad : FB_DoublingTrigger;
	fbHMI_SP_Alarm			: ARRAY[1..DB.MAX_NUMBER_ST] OF FB_HMI_SP_Alarm;
	MSSQL_TcSourceInfo	: ARRAY[1..DB.MAX_NUMBER_ST] OF FB_TcSourceInfo;
	TcEventLogger 	: FB_TcEventLogger;
	RTRIG_BatchChange			: R_TRIG;
END_VAR

fbGetCurTaskIndex();

A_00_Init();
A_10_DiagnosticTools();	// Windows Software tools
A_20_Production();
A_30_SystemTime();
A_92_HMI_Output();
A_99_Alarm();

PRG_EventManagement();

ACTION A_00_Init:
IF _TaskInfo[fbGetCurTaskIndex.index].FirstCycle THEN	// First cycle of this task
	A_99_Alarm_Init();
END_IF
END_ACTION

ACTION A_10_DiagnosticTools:
//UPS Management
PF_00_UPS();

// Launch utility software
NT_CNCScreenDisplay(
	NETID:= '', 
	PATHSTR:= 'C:\Program Files (x86)\CNCScreenE\CNCScrnE.exe', 
	DIRNAME:= '', 
	COMNDLINE:= '', 
	START:= HMI.In.Tools.CNCScreenDisplay, 
	TMOUT:= , 
	BUSY=> HMI.Out.Tools.CNCScreenDisplay, 
	ERR=> , 
	ERRID=> );
	
NT_ProgramTransferTool(
	NETID:= '', 
	PATHSTR:= 'C:\Program Files (x86)\FANUC\Program Transfer Tool\Bin\PttMain.exe', 
	DIRNAME:= '', 
	COMNDLINE:= , 
	START:= HMI.In.Tools.ProgramTransferTool, 
	TMOUT:= , 
	BUSY=> HMI.Out.Tools.ProgramTransferTool, 
	ERR=> , 
	ERRID=> );
	
NT_TaskManager(
	NETID:= , 
	PATHSTR:= 'C:\Windows\system32\Taskmgr.exe', 
	DIRNAME:= '', 
	COMNDLINE:= , 
	START:= HMI.In.Tools.TaskManager, 
	TMOUT:= , 
	BUSY=> HMI.Out.Tools.TaskManager, 
	ERR=> , 
	ERRID=> );
	
NT_OnScreenKeyboard(
	NETID:= , 
	PATHSTR:= 'C:\GSCNext\osk1.bat', 
	DIRNAME:= '', 
	COMNDLINE:= , 
	START:= HMI.In.Tools.OnScreenKeyboard, 
	TMOUT:= , 
	BUSY=> HMI.Out.Tools.OnScreenKeyboard, 
	ERR=> , 
	ERRID=> );
	
NT_CloseBrowser(
	NETID:= , 
	PATHSTR:= 'C:\GSCNext\CloseBrowser.bat', 
	DIRNAME:= '', 
	COMNDLINE:= , 
	START:= HMI.In.Tools.CloseBrowser, 
	TMOUT:= , 
	BUSY=> HMI.Out.Tools.CloseBrowser, 
	ERR=> , 
	ERRID=> );
	
NT_FanucLadder(
	NETID:= , 
	PATHSTR:= 'C:\PROGRAM Files (x86)\FANUC PMC Programmer\FANUC LADDER-3\Fladder.exe', 
	DIRNAME:= '', 
	COMNDLINE:= , 
	START:= HMI.In.Tools.FanucLadder, 
	TMOUT:= , 
	BUSY=> HMI.Out.Tools.FanucLadder, 
	ERR=> , 
	ERRID=> );
	
NT_FlyCad(
	NETID:= , 
	PATHSTR:= 'C:\Program Files (x86)\FlyCAD\flycad.exe', 
	DIRNAME:= '', 
	COMNDLINE:= , 
	START:= HMI.In.Tools.FlyCad, 
	TMOUT:= , 
	BUSY=> HMI.Out.Tools.FlyCad, 
	ERR=> , 
	ERRID=> );

NT_OpenExe( 
	NETID := , 
	PATHSTR := 'C:\GSCNext\UtilityBAT\AperturaExeFromPlc.bat', 
	DIRNAME := 'C:\GSCNext\UtilityBAT', 
	COMNDLINE := , 
	START := , 
	TMOUT := T#5S, 
	BUSY => , 
	ERR => , 
	ERRID =>
);

NT_CloseExe(
	NETID:= , 
	PATHSTR := 'C:\GSCNext\UtilityBAT\ChiusuraExeFromPlc.bat', 
	DIRNAME := 'C:\GSCNext\UtilityBAT', 
	COMNDLINE := , 
	START := , 
	TMOUT := T#5S, 
	BUSY => , 
	ERR => , 
	ERRID => 
);
	
///////////////////////////////////////////////////////////////
TON_OpenPage(IN:= HMI.In.Tools.OpenPage, PT:= T#5S);
HMI.Out.Tools.OpenPage := TON_OpenPage.Q;

///////////////////////////////////////////////////////////////
END_ACTION

ACTION A_20_Production:
fbDoublingTriggerGood(TriggerIn := G.OEE_bCountUpGood);
fbDoublingTriggerBad(TriggerIn := G.OEE_bCountUpBad);

PRG_OEE(Enable := HMI.In.Statistics.OEE_Enable,
		Reset := HMI.In.Statistics.OEE_Reset,
		StartTimer := NOT G.MachineEmpty AND NOT PRG_OEE.Reset,
		bStatusON := HMI.Out.Header.MachineState = eState.Running,
		bStatusOFF := NOT PRG_OEE.bStatusON AND NOT PRG_OEE.bStatusDOWN,
		bStatusDOWN := MachineData.aBool[4],
		tPlannedProductionTime := DWORD_TO_TIME(HMI.Production.OEE.PlannedProductionTime*60000),
		tIdealCycleTime := HMI.Production.OEE.IdealCycleTime,
		bCountUpGood := fbDoublingTriggerGood.TriggerOut,
		bCountUpBad	:= fbDoublingTriggerBad.TriggerOut,
		GoodPieces => HMI.Production.OEE.GoodPieces,
		BadPieces => HMI.Production.OEE.BadPieces,	
);

IF G.OEE_bCountUpGood THEN
	G.OEE_bCountUpGood  := FALSE;
END_IF
IF G.OEE_bCountUpBad THEN
	G.OEE_bCountUpBad  := FALSE;
END_IF

otTON := TIME_TO_OTSTRUCT(PRG_OEE.tON);
otTOFF := TIME_TO_OTSTRUCT(PRG_OEE.tOFF);
otTDOWN := TIME_TO_OTSTRUCT(PRG_OEE.tDOWN);
otTTotal := TIME_TO_OTSTRUCT(PRG_OEE.tON + PRG_OEE.tOFF + PRG_OEE.tDOWN);

HMI.Production.OEE.s_tON 	:= FC_Concat4(WORD_TO_STRING(otTON.wHour) , 'h ',WORD_TO_STRING(otTON.wMinute), 'm');
HMI.Production.OEE.s_tOFF 	:= FC_Concat4(WORD_TO_STRING(otTOFF.wHour) , 'h ',WORD_TO_STRING(otTOFF.wMinute), 'm');
HMI.Production.OEE.s_tDOWN 	:= FC_Concat4(WORD_TO_STRING(otTDOWN.wHour) , 'h ',WORD_TO_STRING(otTDOWN.wMinute), 'm');
HMI.Production.OEE.s_tTOTAL := FC_Concat4(WORD_TO_STRING(otTTotal.wHour) , 'h ',WORD_TO_STRING(otTTotal.wMinute), 'm');

HMI.Production.OEE.Availabilty 	:= 100* PRG_OEE.Availabilty;
HMI.Production.OEE.Performance 	:= 100* PRG_OEE.Performance;
HMI.Production.OEE.Quality 		:= 100* PRG_OEE.Quality;
HMI.Production.OEE.Availabilty 	:= 100* PRG_OEE.Availabilty;
HMI.Production.OEE.OEE 			:= 100* PRG_OEE.OEE;

TempTime1 := TIME_TO_REAL(PRG_OEE.tDOWN);
TempTime2 := TIME_TO_REAL(PRG_OEE.tOFF);
TempTime3 := TIME_TO_REAL(PRG_OEE.tON);
TempSum	:= TempTime1 + TempTime2 + TempTime3;

HMI.Production.OEE.tDOWN := SEL(TempSum <> 0, 0, (TempTime1/TempSum)*100);
HMI.Production.OEE.tOFF	 := SEL(TempSum <> 0, 0, (TempTime2/TempSum)*100);
HMI.Production.OEE.tON	 := SEL(TempSum <> 0, 0, (TempTime3/TempSum)*100);
END_ACTION

ACTION A_30_SystemTime:
GetTime();
IF GetTime.bValid THEN
	G.SystemTime := SYSTEMTIME_TO_DT(GetTime.systemTime);
ELSE
	MEMSET(ADR(G.SystemTime), 16#0, SIZEOF(G.SystemTime));
END_IF
END_ACTION

ACTION A_92_HMI_Output:
// ip definition for user management
HMI.Out.IpDevices[0].Ip := '127.0.0.1';
HMI.Out.IpDevices[0].DeviceType := eDeviceType.Primary;
HMI.Out.IpDevices[1].Ip := '192.168.1.211';
HMI.Out.IpDevices[1].DeviceType := eDeviceType.Secondary;

// BOOL
IF MachineData.aBool[1] THEN
	HMI.Out.Header.OperatingMode := eMode.MODE_SINGLE;
ELSIF MachineData.aBool[0] THEN
	HMI.Out.Header.OperatingMode := eMode.MODE_AUTO;
ELSIF MachineData.aBool[2] THEN
	HMI.Out.Header.OperatingMode := eMode.MODE_MANUAL;
ELSIF MachineData.aBool[5] THEN
	HMI.Out.Header.OperatingMode := eMode.MODE_MAINTENANCE;	
END_IF

IF HMI.Out.UPSDiagnostic.State.ePowerStatus <> E_UpsPowerStatus.PowerOnLine THEN
	HMI.Out.Header.MachineState := eState.UpsOn;
ELSE
	IF MachineData.aBool[7] THEN
		HMI.Out.Header.MachineState := eState.PowerOff;
	ELSIF MachineData.aBool[10] THEN	
		HMI.Out.Header.MachineState := eState.Home;
	ELSIF MachineData.aBool[2] THEN
		HMI.Out.Header.MachineState := eState.Manual;
	ELSIF MachineData.aBool[6] THEN
		HMI.Out.Header.MachineState	:= eState.Ready;
	ELSIF MachineData.aBool[3] THEN
		HMI.Out.Header.MachineState := eState.Running;
	ELSIF MachineData.aBool[4] THEN
		HMI.Out.Header.MachineState := eState.Alarm;
	ELSIF MachineData.aBool[8] THEN
		HMI.Out.Header.MachineState := eState.Emptying;
	ELSIF MachineData.aBool[9] THEN
		HMI.Out.Header.MachineState := eState.Loading;
	ELSE
		HMI.Out.Header.MachineState := eState.Undefine;
	END_IF
END_IF

HMI.Out.Header.Icons[eIcon.Emg] 		:= NOT MachineData.aBool[40];
HMI.Out.Header.Icons[eIcon.DoorOpen] 	:= NOT MachineData.aBool[41];
HMI.Out.Header.Icons[eIcon.AirOk] 		:= MachineData.aBool[42];
HMI.Out.Header.Icons[eIcon.HydraulicOk] := MachineData.aBool[43];
HMI.Out.Header.Icons[eIcon.EquipmentOk] := MachineData.aBool[44];
HMI.Out.Header.Icons[eIcon.Home] 		:= MachineData.aBool[45];
HMI.Out.Header.Icons[eIcon.Connection] 	:= EtherCAT_DevState = 0 AND ProfiNET_DevState = 0 	;
//										   AND MATDiagnostic_MB3000.Running 	AND NOT MATDiagnostic_MB3000.Error
//										   AND MATDiagnostic_MB3500.Running 	AND NOT MATDiagnostic_MB3500.Error
//										   AND MATDiagnostic_MB14000.Running 	AND NOT MATDiagnostic_MB14000.Error	
//										   AND MATDiagnostic_MB14500.Running	AND NOT MATDiagnostic_MB14500.Error		
//										   AND MATDiagnostic_MB8000.Running  	AND NOT MATDiagnostic_MB8000.Error;
										   //AND MATDIAgnostic_MB11000.Running  AND NOT MATDIAgnostic_MB11000.Error
										   //AND MATDiagnostic_MB10600.Running  AND NOT MATDiagnostic_MB10600.Error;

// BYTE
HMI.Out.Header.OvrMultiplier := UINT_TO_STRING(MachineData.aByte[3]);
HMI.Out.Header.PathActive := UINT_TO_STRING(MachineData.aByte[4]);

TON_OvrMultFeedback(PT:=T#300ms);
IF OvrMultiplierOld <> MachineData.aByte[3] THEN
	HMI.Out.Header.OvrMultFeedback := TRUE;
	TON_OvrMultFeedback.IN := TRUE;
	OvrMultiplierOld := MachineData.aByte[3];
END_IF
IF TON_OvrMultFeedback.Q THEN
	HMI.Out.Header.OvrMultFeedback := FALSE;
	TON_OvrMultFeedback.IN := FALSE;
END_IF		

// WORD
HMI.Out.Header.Override := UINT_TO_STRING(MachineData.aWord[0]);
HMI.Out.Header.Feedrate := UINT_TO_STRING(MachineData.aWord[1]); 
HMI.Out.Header.Pieces[eHeaderPieces.Loaded]	:= MachineData.aWord[10];

HMI.Out.Header.Pieces[eHeaderPieces.Total] := SEL(G.MachineEmpty, FC_HeaderCounters(HMI.ShiftData[1].ProcessingData.RunningNoOverRowQty, FALSE),
													FC_HeaderCounters(HMI.ShiftData[17].ProcessingData.RunningNoOverRowQty, FALSE)
												);
												
RTRIG_BatchChange(CLK := G.Batch_old <> HMI.ShiftData[1].ProcessingData.BatchName AND HMI.ShiftData[1].ProcessingData.BatchName <> '');
IF RTRIG_BatchChange.Q THEN
	HMI.Out.Header.Pieces[eHeaderPieces.Ko] := 0;
	HMI.Out.Header.Pieces[eHeaderPieces.Ok] := 0;
	G.Batch_old := HMI.ShiftData[1].ProcessingData.BatchName;
END_IF
HMI.Out.Header.ProgressBar := SEL(HMI.Out.Header.Pieces[eHeaderPieces.Ok] > 0 AND HMI.Out.Header.Pieces[eHeaderPieces.Total] > 0, 0, 
								REAL_TO_USINT((HMI.Out.Header.Pieces[eHeaderPieces.Ok]/UDINT_TO_REAL(HMI.Out.Header.Pieces[eHeaderPieces.Total]))*100.0)
								);

HMI.Out.CycleTime := FC_CycleTimeToString(MAIN.CycleTime);

// Station Status
// -1: alarm
// 0: disabilitata
// 1: home
// 2: working
// 3: home end of job
// 4: unknown
// 5: ciclo estrazione
// 6: ciclo di alimentazione
HMI.St1.Status  := MachineData.aSt[1].State;
HMI.St2.Status  := MachineData.aSt[2].State;
HMI.St3.Status  := MachineData.aSt[3].State;
HMI.St4.Status  := MachineData.aSt[4].State;
HMI.St5.Status  := MachineData.aSt[5].State;
HMI.St6.Status  := MachineData.aSt[6].State;
HMI.St7.Status  := MachineData.aSt[7].State;
HMI.St8.Status  := MachineData.aSt[8].State;
HMI.St9.Status  := MachineData.aSt[9].State;
HMI.St10.Status := MachineData.aSt[10].State;
HMI.St11.Status := MachineData.aSt[11].State;
HMI.St12.Status := MachineData.aSt[12].State;
HMI.St13.Status := MachineData.aSt[13].State;

// Product Status
FOR i := 1 TO NUM_STATIONS + 5 DO
	HMI.ShiftData[i].FLAGP.aByte := MachineData.aSt[i].FlagP_B0;
END_FOR

HMI.St1.ProductStatus  := FC_ProductStatus(HMI.ShiftData[1].FLAGP);
HMI.St2.ProductStatus  := FC_ProductStatus(HMI.ShiftData[2].FLAGP);

IF HMI.St3.TON_DelayProductStatus.Q THEN
	HMI.St3.TON_DelayProductStatus.IN := FALSE;
END_IF
HMI.St3.RTRIG_ProductStatus(CLK := FC_ProductStatus(HMI.ShiftData[3].FLAGP) = eProductStatus.NotPresent);
IF HMI.St3.RTRIG_ProductStatus.Q AND NOT HMI.St3.TON_DelayProductStatus.IN THEN
	HMI.St3.TON_DelayProductStatus.IN := TRUE;
END_IF
HMI.St3.TON_DelayProductStatus(PT := T#1000MS);
IF FC_ProductStatus(HMI.ShiftData[3].FLAGP) <> eProductStatus.NotPresent OR HMI.St3.TON_DelayProductStatus.Q THEN
	HMI.St3.ProductStatus  := FC_ProductStatus(HMI.ShiftData[3].FLAGP);
END_IF

HMI.St4.ProductStatus  := FC_ProductStatus(HMI.ShiftData[4].FLAGP);
HMI.St5.ProductStatus  := FC_ProductStatus(HMI.ShiftData[5].FLAGP);
HMI.St6.ProductStatus  := FC_ProductStatus(HMI.ShiftData[6].FLAGP);
HMI.St7.ProductStatus  := FC_ProductStatus(HMI.ShiftData[7].FLAGP);
HMI.St8.ProductStatus  := FC_ProductStatus(HMI.ShiftData[8].FLAGP);

IF HMI.St9.TON_DelayProductStatus.Q THEN
	HMI.St9.TON_DelayProductStatus.IN := FALSE;
END_IF
HMI.St9.RTRIG_ProductStatus(CLK := FC_ProductStatus(HMI.ShiftData[9].FLAGP) = eProductStatus.NotPresent);
IF HMI.St9.RTRIG_ProductStatus.Q AND NOT HMI.St9.TON_DelayProductStatus.IN THEN
	HMI.St9.TON_DelayProductStatus.IN := TRUE;
END_IF
HMI.St9.TON_DelayProductStatus(PT := T#1000MS);
IF FC_ProductStatus(HMI.ShiftData[9].FLAGP) <> eProductStatus.NotPresent OR HMI.St9.TON_DelayProductStatus.Q THEN
	HMI.St9.ProductStatus  := FC_ProductStatus(HMI.ShiftData[9].FLAGP);
END_IF

HMI.St10.ProductStatus := FC_ProductStatus(HMI.ShiftData[10].FLAGP);
HMI.St11.ProductStatus := FC_ProductStatus(HMI.ShiftData[11].FLAGP);
HMI.St12.ProductStatus := FC_ProductStatus(HMI.ShiftData[12].FLAGP);
HMI.St13.ProductStatus := FC_ProductStatus(HMI.ShiftData[13].FLAGP);
HMI.St14.ProductStatus := FC_ProductStatus(HMI.ShiftData[14].FLAGP);

//processing data
HMI.ProcessingData[1].ProductStatus	:= HMI.St1.ProductStatus;
HMI.ProcessingData[2].ProductStatus	:= HMI.St2.ProductStatus;
HMI.ProcessingData[3].ProductStatus	:= HMI.St3.ProductStatus;
HMI.ProcessingData[4].ProductStatus	:= HMI.St4.ProductStatus;
HMI.ProcessingData[5].ProductStatus	:= HMI.St5.ProductStatus;
HMI.ProcessingData[6].ProductStatus	:= HMI.St6.ProductStatus;
HMI.ProcessingData[7].ProductStatus	:= HMI.St7.ProductStatus;
HMI.ProcessingData[8].ProductStatus	:= HMI.St8.ProductStatus;
HMI.ProcessingData[9].ProductStatus	:= HMI.St9.ProductStatus;
HMI.ProcessingData[10].ProductStatus := HMI.St10.ProductStatus;
HMI.ProcessingData[11].ProductStatus := HMI.St11.ProductStatus;
HMI.ProcessingData[12].ProductStatus := HMI.St12.ProductStatus;
HMI.ProcessingData[13].ProductStatus := HMI.St13.ProductStatus;
HMI.ProcessingData[14].ProductStatus := HMI.St14.ProductStatus;

HMI.ProcessingData[0].Name := TO_STRING(0);
FOR i := 1 TO CNC.NUM_DATA_POSITION DO
	// Assegna dati prodotto o default
	HMI.ProcessingData[i].Name := TO_STRING(i);
	IF HMI.ProcessingData[i].ProductStatus <> eProductStatus.NotPresent THEN
		HMI.ProcessingData[i].PartId                	:= HMI.ShiftData[i].WIDP;
		HMI.ProcessingData[i].ProductName           	:= HMI.ShiftData[i].ProcessingData.ProductName;
		HMI.ProcessingData[i].BatchName 				:= HMI.ShiftData[i].ProcessingData.BatchName; 			
		HMI.ProcessingData[i].RowIndex				    := HMI.ShiftData[i].ProcessingData.RowIndex;			
		HMI.ProcessingData[i].RowRunningNo    		    := HMI.ShiftData[i].ProcessingData.RowRunningNo;   
		HMI.ProcessingData[i].RowQty          		    := HMI.ShiftData[i].ProcessingData.RowQty;        
		HMI.ProcessingData[i].OrderReference  		    := HMI.ShiftData[i].ProcessingData.OrderReference; 
		HMI.ProcessingData[i].Profile     	    		:= HMI.ShiftData[i].ProcessingData.Profile;
		HMI.ProcessingData[i].PlugType	     			:= HMI.ShiftData[i].ProcessingData.PlugType;     
		HMI.ProcessingData[i].Brushing    	    		:= HMI.ShiftData[i].ProcessingData.Brushing;     
		HMI.ProcessingData[i].ProfileLaser	    		:= HMI.ShiftData[i].ProcessingData.ProfileLaser;        
		HMI.ProcessingData[i].BackHole    	    		:= HMI.ShiftData[i].ProcessingData.BackHole;        
		HMI.ProcessingData[i].UnloadMode 		    	:= HMI.ShiftData[i].ProcessingData.UnloadMode;        
		HMI.ProcessingData[i].RunningNoOverRowQty 		:= HMI.ShiftData[i].ProcessingData.RunningNoOverRowQty;
		//HMI.ProcessingData[i].CurrentRowOverRowCount 	:= HMI.ShiftData[i].ProcessingData.CurrentRowOverRowCount;
	ELSE
		HMI.ProcessingData[i].PartId                	:= 0;
		HMI.ProcessingData[i].ProductName           	:= '';
		HMI.ProcessingData[i].BatchName 				:= '';	
		HMI.ProcessingData[i].RowIndex					:= '';
		HMI.ProcessingData[i].RowRunningNo    			:= '';
		HMI.ProcessingData[i].RowQty          			:= '';
		HMI.ProcessingData[i].OrderReference  			:= '';
		HMI.ProcessingData[i].Profile     	    		:= '';
		HMI.ProcessingData[i].PlugType	     			:= '';
		HMI.ProcessingData[i].Brushing    	    		:= '';
		HMI.ProcessingData[i].ProfileLaser	    		:= '';
		HMI.ProcessingData[i].BackHole    	    		:= '';
		HMI.ProcessingData[i].UnloadMode 		    	:= '';
		HMI.ProcessingData[i].RunningNoOverRowQty 		:= '';
		HMI.ProcessingData[i].CurrentRowOverRowCount	:= '';
	END_IF	
END_FOR

fbRefresh(bRefreshHMI := HMI.Out.ProductionQueueRefresh);
END_ACTION

ACTION A_99_Alarm:
RTRIG_ClearAlarm(CLK := G.ResetButton);
IF RTRIG_ClearAlarm.Q THEN
	M_98_Marker_AlarmClear();
	M_98_DataRequest_AlarmClear();
	M_98_MSSQL_AlarmClear();
END_IF

TON_DelayMarkerConnected(IN := MAIN.Lasit.bEnable AND NOT MAIN.Lasit.bConnected, PT := T#10S);
M_99_Marker_Alarm();
M_99_DataRequest_Alarm();
M_99_MSSQL_Alarm();
END_ACTION

ACTION A_99_Alarm_Init:
TcSourceInfo.sName := 'PLC';

M_00_Init_Marker_Alarm();
M_00_Init_DataRequest_Alarm();
M_00_Init_MSSQL_Alarm();
END_ACTION

METHOD PRIVATE M_00_Init_DataRequest_Alarm
DataRequest_Events.aAlarm[0].CreateEx(TC_Events.DataRequest_Alarm.A80000,FALSE,TcSourceInfo);
DataRequest_Events.aAlarm[1].CreateEx(TC_Events.DataRequest_Alarm.A80001,FALSE,TcSourceInfo);
DataRequest_Events.aAlarm[2].CreateEx(TC_Events.DataRequest_Alarm.A80002,FALSE,TcSourceInfo);
DataRequest_Events.aAlarm[3].CreateEx(TC_Events.DataRequest_Alarm.A80003,FALSE,TcSourceInfo);
DataRequest_Events.aAlarm[4].CreateEx(TC_Events.DataRequest_Alarm.A80004,FALSE,TcSourceInfo);
DataRequest_Events.aAlarm[5].CreateEx(TC_Events.DataRequest_Alarm.A80005,FALSE,TcSourceInfo);
END_METHOD

METHOD PRIVATE M_00_Init_Marker_Alarm
Marker_Events.aAlarm[0].CreateEx(TC_Events.Marker_Alarm.A60000,FALSE,TcSourceInfo);
Marker_Events.aAlarm[1].CreateEx(TC_Events.Marker_Alarm.A60001,FALSE,TcSourceInfo);
Marker_Events.aAlarm[2].CreateEx(TC_Events.Marker_Alarm.A60002,FALSE,TcSourceInfo);
Marker_Events.aAlarm[3].CreateEx(TC_Events.Marker_Alarm.A60003,FALSE,TcSourceInfo);
Marker_Events.aAlarm[4].CreateEx(TC_Events.Marker_Alarm.A60004,FALSE,TcSourceInfo);
Marker_Events.aAlarm[5].CreateEx(TC_Events.Marker_Alarm.A60005,FALSE,TcSourceInfo);
Marker_Events.aAlarm[6].CreateEx(TC_Events.Marker_Alarm.A60006,FALSE,TcSourceInfo);

Marker_Events.aAlarm[10].CreateEx(TC_Events.Marker_Alarm.A60010,FALSE,TcSourceInfo);
Marker_Events.aAlarm[11].CreateEx(TC_Events.Marker_Alarm.A60011,FALSE,TcSourceInfo);
Marker_Events.aAlarm[12].CreateEx(TC_Events.Marker_Alarm.A60012,FALSE,TcSourceInfo);
Marker_Events.aAlarm[13].CreateEx(TC_Events.Marker_Alarm.A60013,FALSE,TcSourceInfo);
END_METHOD

METHOD PRIVATE M_00_Init_MSSQL_Alarm
MSSQL_Events.aAlarm[0].CreateEx(TC_Events.DB_Alarm.A50000,FALSE,TcSourceInfo);
MSSQL_Events.aAlarm[1].CreateEx(TC_Events.DB_Alarm.A50001,FALSE,TcSourceInfo);
MSSQL_Events.aAlarm[2].CreateEx(TC_Events.DB_Alarm.A50002,FALSE,TcSourceInfo);
MSSQL_Events.aAlarm[3].CreateEx(TC_Events.DB_Alarm.A50003,FALSE,TcSourceInfo);

MSSQL_Events.aAlarm[10].CreateEx(TC_Events.DB_Alarm.A50010,FALSE,TcSourceInfo);
MSSQL_Events.aAlarm[11].CreateEx(TC_Events.DB_Alarm.A50011,FALSE,TcSourceInfo);
MSSQL_Events.aAlarm[12].CreateEx(TC_Events.DB_Alarm.A50012,FALSE,TcSourceInfo);
MSSQL_Events.aAlarm[13].CreateEx(TC_Events.DB_Alarm.A50013,FALSE,TcSourceInfo);

MSSQL_Events.aAlarm[20].CreateEx(TC_Events.DB_Alarm.A50020,FALSE,TcSourceInfo);
MSSQL_Events.aAlarm[21].CreateEx(TC_Events.DB_Alarm.A50021,FALSE,TcSourceInfo);
MSSQL_Events.aAlarm[22].CreateEx(TC_Events.DB_Alarm.A50022,FALSE,TcSourceInfo);
MSSQL_Events.aAlarm[23].CreateEx(TC_Events.DB_Alarm.A50023,FALSE,TcSourceInfo);
                                                                 
MSSQL_Events.aAlarm[30].CreateEx(TC_Events.DB_Alarm.A50030,FALSE,TcSourceInfo);
MSSQL_Events.aAlarm[31].CreateEx(TC_Events.DB_Alarm.A50031,FALSE,TcSourceInfo);
MSSQL_Events.aAlarm[32].CreateEx(TC_Events.DB_Alarm.A50032,FALSE,TcSourceInfo);
MSSQL_Events.aAlarm[33].CreateEx(TC_Events.DB_Alarm.A50033,FALSE,TcSourceInfo);
MSSQL_Events.aAlarm[34].CreateEx(TC_Events.DB_Alarm.A50034,FALSE,TcSourceInfo);
MSSQL_Events.aAlarm[35].CreateEx(TC_Events.DB_Alarm.A50035,FALSE,TcSourceInfo);
                                                                 
MSSQL_Events.aAlarm[40].CreateEx(TC_Events.DB_Alarm.A50040,FALSE,TcSourceInfo);
MSSQL_Events.aAlarm[41].CreateEx(TC_Events.DB_Alarm.A50041,FALSE,TcSourceInfo);
MSSQL_Events.aAlarm[42].CreateEx(TC_Events.DB_Alarm.A50042,FALSE,TcSourceInfo);
END_METHOD

METHOD PRIVATE M_98_DataRequest_AlarmClear
VAR
	i :UINT := 0;
	j :UINT := 0;
END_VAR
FOR j := 0 TO G.MAX_ALR_WORD DO
	IF DataRequest_Events.wAlarm[j]<> 0 THEN
		FOR i:= 0 TO G.MAX_ALR DO
			DataRequest_Events.aAlarm[i].Clear(0,TRUE);			
		END_FOR	
	END_IF
	DataRequest_Events.wAlarm[j] := 0;
END_FOR
END_METHOD

METHOD PRIVATE M_98_Marker_AlarmClear
VAR
	i :UINT := 0;
	j :UINT := 0;
END_VAR
FOR j := 0 TO G.MAX_ALR_WORD DO
	IF Marker_Events.wAlarm[j]<> 0 THEN
		FOR i:= 0 TO G.MAX_ALR DO
			Marker_Events.aAlarm[i].Clear(0,TRUE);			
		END_FOR	
	END_IF
	Marker_Events.wAlarm[j] := 0;
END_FOR
END_METHOD

METHOD PRIVATE M_98_MSSQL_AlarmClear
VAR
	i :UINT := 0;
	j :UINT := 0;
END_VAR
FOR j := 0 TO G.MAX_ALR_WORD DO
	IF MSSQL_Events.wAlarm[j]<> 0 THEN
		FOR i:= 0 TO G.MAX_ALR DO
			MSSQL_Events.aAlarm[i].Clear(0,TRUE);			
		END_FOR	
	END_IF
	MSSQL_Events.wAlarm[j] := 0;
END_FOR
END_METHOD

METHOD PRIVATE M_99_DataRequest_Alarm
VAR
	i :UINT := 0;
END_VAR
DataRequest_Events.Cumulative := FALSE;
FOR i := 0 TO G.MAX_ALR_WORD DO
	IF DataRequest_Events.wAlarm[i]<> 0 THEN
		DataRequest_Events.Cumulative := TRUE;
		EXIT;
	END_IF
END_FOR

IF MAIN.fbDataRequest.Error THEN
	CASE MAIN.fbDataRequest.ErrorID OF
		1020://fbDataRequest - GetNextPLCData error
			DataRequest_Events.wAlarm[0].2 := 1;
			DataRequest_Events.aAlarm[2].Raise(0);
		1031:// errore stringa abilitazione foro coda (non rispetta le impostazioni)
			DataRequest_Events.wAlarm[0].4 := 1;
			DataRequest_Events.aAlarm[4].Raise(0); 
		1032:// errore stringa abilitazione foro coda (vuota)
			DataRequest_Events.wAlarm[0].5 := 1;
			DataRequest_Events.aAlarm[5].Raise(0);
		1999://fbDataRequest - Timeout
			DataRequest_Events.wAlarm[0].1 := 1;
			DataRequest_Events.aAlarm[1].ipArguments.Clear().AddDInt(MAIN.fbDataRequest.ErrorSubID);
			DataRequest_Events.aAlarm[1].Raise(0);
		ELSE///fbDataRequest - Generic error
			IF MAIN.fbDataRequest.ErrorID <> 1030 THEN
				DataRequest_Events.wAlarm[0].0 := 1;
				DataRequest_Events.aAlarm[0].ipArguments.Clear().AddDInt(MAIN.fbDataRequest.ErrorID);
				DataRequest_Events.aAlarm[0].Raise(0);	
			END_IF
	END_CASE
END_IF
END_METHOD

METHOD PRIVATE M_99_Marker_Alarm
VAR
	i :UINT := 0;
END_VAR
Marker_Events.Cumulative := FALSE;
FOR i := 0 TO G.MAX_ALR_WORD DO
	IF Marker_Events.wAlarm[i]<> 0 THEN
		Marker_Events.Cumulative := TRUE;
		EXIT;
	END_IF
END_FOR	

IF TON_DelayMarkerConnected.Q THEN
	Marker_Events.wAlarm[0].2 := 1;
	Marker_Events.aAlarm[2].Raise(0);
END_IF

IF MAIN.LasitManager.Error THEN
	CASE MAIN.LasitManager.ErrorID OF
		1000:// lasit not connected
			Marker_Events.wAlarm[0].3 := 1;
			Marker_Events.aAlarm[3].Raise(0);
		1010:// lasit not found layout in the list	
			Marker_Events.wAlarm[0].4 := 1;
			Marker_Events.aAlarm[4].Raise(0);
		1030:// lasit loading layout error
			Marker_Events.wAlarm[0].5 := 1;
			Marker_Events.aAlarm[5].Raise(0);
		1070:// lasit loading text error
			Marker_Events.wAlarm[0].6 := 1;
			Marker_Events.aAlarm[6].Raise(0);
		1999://fbDataRequest - Timeout
			Marker_Events.wAlarm[0].1 := 1;
			Marker_Events.aAlarm[1].ipArguments.Clear().AddDInt(MAIN.LasitManager.ErrorSubID);
			Marker_Events.aAlarm[1].Raise(0);
		ELSE// lasit generic error
			Marker_Events.wAlarm[0].0 := 1;
			Marker_Events.aAlarm[0].ipArguments.Clear().AddDInt(MAIN.LasitManager.ErrorID);
			Marker_Events.aAlarm[0].Raise(0);
	END_CASE
END_IF

IF MAIN.fbFlyPowerMarkExeManager.Error THEN
	CASE MAIN.fbFlyPowerMarkExeManager.ErrorID OF
		1030:// powermark error tentativo di apertura fallito
			Marker_Events.wAlarm[0].12 := 1;
			Marker_Events.aAlarm[12].Raise(0);
		1020:// powermark error tentativo di chiusura fallito
			Marker_Events.wAlarm[0].13 := 1;
			Marker_Events.aAlarm[13].Raise(0);
		1999://powermark error - Timeout
			Marker_Events.wAlarm[0].11 := 1;
			Marker_Events.aAlarm[11].ipArguments.Clear().AddDInt(MAIN.fbFlyPowerMarkExeManager.ErrorSubID);
			Marker_Events.aAlarm[11].Raise(0);
		ELSE// powermark generic error
			Marker_Events.wAlarm[10].0 := 1;
			Marker_Events.aAlarm[10].ipArguments.Clear().AddDInt(MAIN.fbFlyPowerMarkExeManager.ErrorID);
			Marker_Events.aAlarm[10].Raise(0);
	END_CASE
END_IF
END_METHOD

METHOD PRIVATE M_99_MSSQL_Alarm
VAR
	i :UDINT := 0;
END_VAR
MSSQL_Events.Cumulative := FALSE;
FOR i := 0 TO G.MAX_ALR_WORD DO
	IF MSSQL_Events.wAlarm[i]<> 0 THEN
		MSSQL_Events.Cumulative := TRUE;
		EXIT;
	END_IF
END_FOR

IF PRG_MSSQL_InitConnection.Error THEN
	CASE PRG_MSSQL_InitConnection.ErrorID OF
		
		1001:// connection error
			MSSQL_Events.wAlarm[0].1 := 1;
			MSSQL_Events.aAlarm[1].Raise(0);
			
		1003:// disconnection error
			MSSQL_Events.wAlarm[0].2 := 1;
			MSSQL_Events.aAlarm[2].Raise(0);
			
		1010, 1020, 1030, 1040:// init sql commands error
			MSSQL_Events.wAlarm[0].3 := 1;
			MSSQL_Events.aAlarm[3].ipArguments.Clear().AddDInt(PRG_MSSQL_InitConnection.ErrorID);
			MSSQL_Events.aAlarm[3].Raise(0);
			
		ELSE// init sql stored procedure error
			MSSQL_Events.wAlarm[0].0 := 1;
			MSSQL_Events.aAlarm[0].ipArguments.Clear().AddDInt(PRG_MSSQL_InitConnection.ErrorID);
			MSSQL_Events.aAlarm[0].Raise(0);
	END_CASE
END_IF

///////////////////////////////////////////////////////////////
IF PRG_MSSQL_spGetNextPartPLCData.Error THEN
	CASE PRG_MSSQL_spGetNextPartPLCData.ErrorID OF
		
		1050://Req new PLC data execute error
			MSSQL_Events.wAlarm[1].1 := 1;
			MSSQL_Events.aAlarm[11].Raise(0);
			
		1060://Req new PLC data read error
			MSSQL_Events.wAlarm[1].2 := 1;
			MSSQL_Events.aAlarm[12].Raise(0);
			
		1080://Req new PLC data result conversion error
			MSSQL_Events.wAlarm[1].3 := 1;
			MSSQL_Events.aAlarm[13].ipArguments.Clear().AddDInt(PRG_MSSQL_spGetNextPartPLCData.ErrorID);
			MSSQL_Events.aAlarm[13].Raise(0);
		
		-10001:// SP on DB generic error
			MSSQL_Events.wAlarm[2].4 := 1;
			MSSQL_Events.aAlarm[14].Raise(0);			
		-10101:// SP on DB Row Not Found
			MSSQL_Events.wAlarm[2].5 := 1;
			MSSQL_Events.aAlarm[15].Raise(0);
		-11001:// SP on DB ProfileNotFound
			MSSQL_Events.wAlarm[2].6 := 1;
			MSSQL_Events.aAlarm[16].Raise(0);
		-11002:// SP on DB BroachNotFound
			MSSQL_Events.wAlarm[2].7 := 1;
			MSSQL_Events.aAlarm[17].Raise(0);
		-11003:// SP on DB InvalidBroachSequence
			MSSQL_Events.wAlarm[2].8 := 1; 
			MSSQL_Events.aAlarm[18].Raise(0);
		-12001:// SP on DB LookUpNameNotFound
			MSSQL_Events.wAlarm[2].9 := 1;
			MSSQL_Events.aAlarm[19].Raise(0);
		ELSE
			IF PRG_MSSQL_spGetNextPartPLCData.ErrorID > 10000 THEN
				// batch state on db undefine	
				MSSQL_Events.wAlarm[2].21 := 1;
				MSSQL_Events.aAlarm[47].Raise(0);
			ELSE
				//Req new PLC data generic error
				MSSQL_Events.wAlarm[1].0 := 1;
				MSSQL_Events.aAlarm[10].ipArguments.Clear().AddDInt(PRG_MSSQL_spGetNextPartPLCData.ErrorID);
				MSSQL_Events.aAlarm[10].Raise(0);
			END_IF
	END_CASE
END_IF

///////////////////////////////////////////////////////////////
IF PRG_MSSQL_UpdatePartLocationsAndProcessingData.Error THEN
	CASE PRG_MSSQL_UpdatePartLocationsAndProcessingData.ErrorID OF
		
		1010://Update processin data conversion error
			MSSQL_Events.wAlarm[2].1 := 1;
			MSSQL_Events.aAlarm[21].Raise(0);
	
		1020://Update processin data execute error
			MSSQL_Events.wAlarm[2].2 := 1;
			MSSQL_Events.aAlarm[22].Raise(0);
		
		ELSE//Update processin data generic error
			MSSQL_Events.wAlarm[2].0 := 1;
			MSSQL_Events.aAlarm[20].ipArguments.Clear().AddDInt(PRG_MSSQL_UpdatePartLocationsAndProcessingData.ErrorID);
			MSSQL_Events.aAlarm[20].Raise(0);
	END_CASE
END_IF

///////////////////////////////////////////////////////////////
IF PRG_MSSQL_spGetProcessingDataForHMI.Error THEN
	CASE PRG_MSSQL_spGetProcessingDataForHMI.ErrorID OF
		
		1010://Get processin data execute error
			MSSQL_Events.wAlarm[3].1 := 1;
			MSSQL_Events.aAlarm[31].Raise(0);
			
		1020://Get processin data read error
			MSSQL_Events.wAlarm[3].2 := 1;
			MSSQL_Events.aAlarm[32].Raise(0);
			
		1040://Get processin data buffer empty
			MSSQL_Events.wAlarm[3].3 := 1;
			MSSQL_Events.aAlarm[33].Raise(0);
			
		1041://Get processin data json conversion error
			MSSQL_Events.wAlarm[3].4 := 1;
			MSSQL_Events.aAlarm[34].Raise(0);
		
		1042://Get processin data json conversion error
			MSSQL_Events.wAlarm[3].5 := 1;
			MSSQL_Events.aAlarm[35].Raise(0);
				
		ELSE//Get processin data generic error
			MSSQL_Events.wAlarm[3].0 := 1;
			MSSQL_Events.aAlarm[30].ipArguments.Clear().AddDInt(PRG_MSSQL_spGetProcessingDataForHMI.ErrorID);
			MSSQL_Events.aAlarm[30].Raise(0);
	END_CASE
END_IF

///////////////////////////////////////////////////////////////
IF PRG_MSSQL_spCMD_AbortProduction.Error THEN
	CASE PRG_MSSQL_spCMD_AbortProduction.ErrorID OF
		
		1010://sp execute error
			MSSQL_Events.wAlarm[4].1 := 1;
			MSSQL_Events.aAlarm[41].Raise(0);
			
		1020://sp failed
			MSSQL_Events.wAlarm[4].2 := 1;
			MSSQL_Events.aAlarm[42].Raise(0);
		
		ELSE//sp generic error
			MSSQL_Events.wAlarm[4].0 := 1;
			MSSQL_Events.aAlarm[40].ipArguments.Clear().AddDInt(PRG_MSSQL_spCMD_AbortProduction.ErrorID);
			MSSQL_Events.aAlarm[40].Raise(0);
	END_CASE
END_IF

//////////////////////////// HMI ///////////////////////////////////

FOR i := 1 TO DB.MAX_NUMBER_ST DO
	fbHMI_SP_Alarm[i](	Error			:= DB.HMI_SP_Alarm[i].Error,	
						ErrorID			:= DB.HMI_SP_Alarm[i].ErrorID,			
						aAlarm			:= ADR(MSSQL_Events.aAlarm[100]),
						wAlarm			:= ADR(MSSQL_Events.wAlarm[10]),
						SourceName		:= CONCAT('SP_', TO_STRING(i)),
						TcSourceInfo	:= MSSQL_TcSourceInfo[i],
						TcEventLogger 	:= TcEventLogger,
						EventId			:= 50100);
END_FOR
END_METHOD

END_PROGRAM

// ---- FBs/FB_RetainTimer.TcPOU
FUNCTION_BLOCK FB_RetainTimer
VAR_INPUT
	Enable 		: BOOL;			// Enable timer
	Reset 		: BOOL;			// Reset timer
END_VAR
VAR_OUTPUT
	ET			: TIME := T#0S;	// Elapsed TIME
	ET_ms		: DWORD;		// Elapsed DWORD milliseconds
END_VAR
VAR
	RTRIG_Enable	: R_TRIG;
	FTRIG_Enable	: F_TRIG;
	RTRIG_Reset		: R_TRIG;
	StartTime		: TIME := T#0S;
	SessionTime		: TIME := T#0S;
	TotalTime		: TIME := T#0S;
END_VAR

RTRIG_Enable(CLK := Enable);
FTRIG_Enable(CLK := Enable);
RTRIG_Reset(CLK := Reset);

// RESET
	IF(RTRIG_Reset.Q) THEN
		StartTime 	:= T#0S;
		SessionTime := T#0S;
		TotalTime 	:= T#0S;
	END_IF

// ENABLE
	IF(RTRIG_Enable.Q AND NOT Reset) THEN
		StartTime := TIME();
	END_IF
	
	IF(FTRIG_Enable.Q) THEN
		TotalTime := TotalTime + SessionTime;
		SessionTime := T#0s;
	END_IF

///////////////////////////////////////////////////////////////

// Updating time
IF(Enable AND NOT Reset) THEN
	SessionTime := TIME() - StartTime;
END_IF

ET := TotalTime + SessionTime;
ET_ms := TIME_TO_DWORD(ET);

END_FUNCTION_BLOCK

// ---- FBs/FB_Refresh.TcPOU
FUNCTION_BLOCK FB_Refresh
VAR_IN_OUT
    bRefreshHMI : BOOL;          // → HMI
END_VAR
VAR
    fbPeriod    : TON := (PT := T#1S);      // Timer periodo di 1 s
    fbWatchdog  : TON := (PT := T#500MS);   // Watch‑dog di 500 ms
    bWaitingForReset : BOOL;                // TRUE finché aspettiamo il reset
END_VAR

(* --- fase di attesa impulso --- *)
IF NOT bWaitingForReset THEN
    fbPeriod(IN := TRUE);                

    IF fbPeriod.Q OR bRefreshHMI THEN                   
        bRefreshHMI := TRUE;             // dico all’HMI “sono vivo”
        fbPeriod(IN := FALSE);           // fermo il period
        fbWatchdog(IN := TRUE);          // start WD (1ª chiamata)
        bWaitingForReset := TRUE;
    END_IF

(* --- fase di attesa reset HMI o watchdog --- *)
ELSE
    fbPeriod(IN := FALSE);               // periodo fermo
    fbWatchdog(IN := TRUE);

    IF NOT bRefreshHMI THEN              // HMI ha resettato
        fbWatchdog(IN := FALSE);         // stop WD
        bWaitingForReset := FALSE;

    ELSIF fbWatchdog.Q THEN              
        bRefreshHMI := FALSE;            // forzo reset
        fbWatchdog(IN := FALSE);         // riarmo
        bWaitingForReset := FALSE;
    END_IF
END_IF

END_FUNCTION_BLOCK

// ---- FBs/FB_DoublingTrigger.TcPOU
FUNCTION_BLOCK FB_DoublingTrigger
VAR_INPUT
    TriggerIn : BOOL; // Segnale di trigger in ingresso
END_VAR
VAR_OUTPUT
    TriggerOut : BOOL; // Unico segnale di uscita, attivo per 1 ciclo due volte
END_VAR
VAR
    TrigPrev : BOOL;
	R_TrigIn : R_TRIG;
    timerDelay : TON;
    state : INT; // 0 = idle, 1 = primo impulso, 2 = attesa 100ms, 3 = secondo impulso
END_VAR

R_TrigIn(CLK := TriggerIn);

// Reset uscita
TriggerOut := FALSE;

CASE state OF
    0: // Attesa trigger
        IF R_TrigIn.Q THEN
            TriggerOut := TRUE; // Primo impulso
            timerDelay(IN := TRUE, PT := T#100ms);
            state := 1;
        END_IF

    1: // Timer in corso
        timerDelay(IN := TRUE);
        IF timerDelay.Q THEN
            timerDelay(IN := FALSE); // Ferma il timer
            TriggerOut := TRUE;     // Secondo impulso
            state := 2;
        END_IF

    2: // Attendi fine ciclo per tornare idle
        state := 0;
END_CASE

END_FUNCTION_BLOCK

// ---- FBs/Database/FB_HMI_SP_Alarm.TcPOU
FUNCTION_BLOCK FB_HMI_SP_Alarm
VAR_INPUT
	Error						: BOOL;
	ErrorID						: DINT;
	aAlarm						: POINTER TO FB_TcAlarm;
	wAlarm						: POINTER TO DWORD;
	SourceName					: STRING;
	TcSourceInfo				: FB_TcSourceInfo;
	TcEventLogger 				: FB_TcEventLogger;
	EventId						: UDINT;
END_VAR
VAR
	bResult : BOOL;
	AlarmExist						: ARRAY[0..G.MAX_ALR] OF BOOL;
END_VAR

bResult := FALSE;
IF Error THEN
	CASE ErrorID OF
		1010://Execute error
			wAlarm^.2 := 1;
			
			IF NOT AlarmExist[2] THEN 
				AlarmExist[2] := TRUE; 
				bResult := FC_AlarmExists(SourceName, TcSourceInfo, TcEventLogger, aAlarm[2], TC_Events.DB_Alarm.A50102, (EventId + 2));
			ELSE 
				bResult := TRUE; 
			END_IF
			
			IF bResult THEN
				aAlarm[2].Raise(0);
			END_IF
		1020://read error
			wAlarm^.3 := 1;
			
			IF NOT AlarmExist[3] THEN 
				AlarmExist[3] := TRUE; 
				bResult := FC_AlarmExists(SourceName, TcSourceInfo, TcEventLogger, aAlarm[3], TC_Events.DB_Alarm.A50103, (EventId + 3));
			ELSE 
				bResult := TRUE; 
			END_IF
			IF bResult THEN
				aAlarm[3].Raise(0);	
			END_IF
		1999://Timeout
			wAlarm^.1 := 1;
			
			IF NOT AlarmExist[1] THEN 
				AlarmExist[1] := TRUE; 
				bResult := FC_AlarmExists(SourceName, TcSourceInfo, TcEventLogger, aAlarm[1], TC_Events.DB_Alarm.A50101, (EventId + 1));
			ELSE 
				bResult := TRUE; 
			END_IF
			IF bResult THEN
				aAlarm[1].Raise(0);
			END_IF
		ELSE // Generic
			wAlarm^.0 := 1;
			
			IF NOT AlarmExist[0] THEN 
				AlarmExist[0] := TRUE; 
				bResult := FC_AlarmExists(SourceName, TcSourceInfo, TcEventLogger, aAlarm[0], TC_Events.DB_Alarm.A50100, (EventId + 0));
			ELSE 
				bResult := TRUE; 
			END_IF
			IF bResult THEN
				aAlarm[0].ipArguments.Clear().AddDInt(ErrorID);
				aAlarm[0].Raise(0);	
			END_IF
	END_CASE
END_IF

END_FUNCTION_BLOCK

// ---- FCs/FC_AlarmExists.TcPOU
FUNCTION FC_AlarmExists : BOOL
VAR_INPUT
    SourceName: STRING(255) := '';
	TcSourceInfo	: FB_TcSourceInfo;
	TcEventLogger 	: FB_TcEventLogger;
	TcAlarm	: REFERENCE TO FB_TcAlarm;
	pTcEventEntry	: TcEventEntry;
	EventId	: UDINT;
END_VAR
VAR
	hr	: HRESULT;
END_VAR

TcSourceInfo.sName := CONCAT('PLC.', SourceName);
hr := TcEventLogger.GetAlarm(pTcEventEntry.uuidEventClass, EventId, TcSourceInfo, TcAlarm);

// Create event if not already created
IF NOT SUCCEEDED(hr) THEN		
	hr := TcAlarm.CreateEx(pTcEventEntry, FALSE, TcSourceInfo);
END_IF;	

IF SUCCEEDED(hr) THEN		
	FC_AlarmExists := TRUE;
ELSE
	FC_AlarmExists := FALSE;
END_IF;

END_FUNCTION

// ---- POUs/PF_00_UPS.TcPOU
PROGRAM PF_00_UPS
VAR
	fbUPS				: FB_GetUPSStatus;
	fbWrite				: FB_WritePersistentData;
	eState				: E_UpsPowerStatus;
	uWriteState			: UINT :=0;
	bWriteOK			: BOOL := FALSE;
	bWriteStart			: BOOL;
	RTRIG_WriteStart	: R_TRIG;
END_VAR

fbUPS(	sNetID	:= '', 
		nPort	:= , 
		bEnable	:= TRUE);

fbWrite(	NETID 	:=,
			PORT	:= 851,
			TMOUT	:= T#20S,
			MODE	:= E_PersistentMode.SPDM_2PASS);

HMI.Out.UPSDiagnostic.Valid := fbUPS.bValid;
			
IF fbUPS.bValid THEN

	eState := fbUPS.stStatus.ePowerStatus;
	
	CASE eState OF
		E_UpsPowerStatus.PowerOnLine:
			IF NOT fbWrite.BUSY THEN
				uWriteState := 0;
				bWriteOK	:= FALSE;
				bWriteStart := FALSE;
			END_IF
			
		E_UpsPowerStatus.PowerOnBattery:
			bWriteStart := TRUE;
			
		E_UpsPowerStatus.PowerUnknownStatus:
			; // error
	
	END_CASE

	HMI.Out.UPSDiagnostic.State := fbUPS.stStatus;	

END_IF	

RTRIG_WriteStart(CLK := bWriteStart);
IF RTRIG_WriteStart.Q THEN
	uWriteState := 10;
END_IF
CASE uWriteState OF
	0:
		;
		
	10:
		fbWrite.START := TRUE;			
		
		uWriteState := 20;
		
	20:
		IF NOT fbWrite.BUSY THEN
			fbWrite.START := FALSE;	
			IF fbWrite.ERR THEN
				
				uWriteState := 1030;
			ELSE
				bWriteOK:= TRUE;
				
				uWriteState := 0;
			END_IF
		END_IF

END_CASE

END_PROGRAM

// ---- POUs/PRG_OEE.TcPOU
PROGRAM PRG_OEE

VAR_INPUT
	Enable					: BOOL;
	Reset					: BOOL;
	StartTimer				: BOOL;
	bStatusON				: BOOL;
	bStatusDOWN				: BOOL;
	bStatusOFF				: BOOL;
	bCountUpGood			: BOOL;
	bCountUpBad				: BOOL;
	tIdealCycleTime			: TIME;
	tPlannedProductionTime	: TIME;
END_VAR

VAR_OUTPUT
	GoodPieces				: DINT := 0;
	BadPieces				: DINT := 0;
	Availabilty 			: REAL	:= 0;
	Performance 			: REAL	:= 0;
	Quality					: REAL	:= 0;
	OEE						: REAL	:= 0;
	tON						: TIME	:= T#0S;
	tOFF					: TIME	:= T#0S;
	tDOWN					: TIME	:= T#0s;
	
END_VAR

VAR
	RTRIG_Reset				: R_TRIG;
	EndSessionTime			: TIME := T#0S;
	iState					: INT := 0;
	RTON_ON					: FB_RetainTimer;
	RTON_OFF				: FB_RetainTimer;
	RTON_DOWN				: FB_RetainTimer;
	RTRIG_StartTimer		: R_TRIG;
	TotalPieces				: UDINT;
	TotalTime_ms			: DWORD;
	rOperatingTime			: REAL;
	rProductionTime			: REAL;
	CTU_GoodPieces			: CTU;
	CTU_BadPieces			: CTU;
	TimeStart				: TIME;
	OperatingTime			: TIME;
END_VAR

RTRIG_StartTimer(CLK := StartTimer);
RTRIG_Reset(CLK := Reset);
IF(RTRIG_Reset.Q) THEN
	iState := 0;
END_IF

// Retain timers
	RTON_ON(Enable := bStatusON AND Enable AND StartTimer AND NOT Reset, Reset := iState = 0, ET => tON);
	RTON_OFF(Enable := bStatusOFF AND Enable AND StartTimer AND NOT Reset, Reset := iState = 0, ET => tOFF);
	RTON_DOWN(Enable := bStatusDOWN AND Enable AND StartTimer AND NOT Reset, Reset := iState = 0, ET => tDOWN);

// CounterUp 
	CTU_GoodPieces(CU := bCountUpGood AND NOT bStatusDOWN, Reset := iState = 10);
	CTU_BadPieces(CU := bCountUpBad AND NOT bStatusDOWN, Reset := iState = 10);


CASE iState OF
	0:
		GoodPieces					:= 0;
		BadPieces					:= 0;
		Performance 				:= 0;
		Availabilty 				:= 0;
		Quality 					:= 0;
		OEE							:= 0;
		
		iState := 10;
		
	10:
		IF(Enable) AND RTRIG_StartTimer.Q THEN
			TimeStart 		:= TIME();
			EndSessionTime 	:= TimeStart + tPlannedProductionTime;

			iState := 20;
		END_IF
	
	20:
		// COUTNERS
			GoodPieces := CTU_GoodPieces.CV;
			BadPieces := CTU_BadPieces.CV;
			
		// AVAILABILITY
			TotalTime_ms := RTON_ON.ET_ms + RTON_OFF.ET_ms + RTON_DOWN.ET_ms;
			IF(TotalTime_ms > 0) THEN
				Availabilty :=  (DWORD_TO_REAL(RTON_ON.ET_ms) + DWORD_TO_REAL(RTON_OFF.ET_ms)) / DWORD_TO_REAL(TotalTime_ms);
			ELSE
				Availabilty := 0;
			END_IF
		
		// QUALITY
			TotalPieces := GoodPieces + BadPieces;
			IF(TotalPieces > 0) THEN
				Quality := TO_REAL(GoodPieces) / TO_REAL(TotalPieces);
			ELSE
				Quality := 0;
			END_IF
			
		// PERFORMANCE
			OperatingTime := RTON_ON.ET + RTON_DOWN.ET;
			IF(TIME_TO_DWORD(OperatingTime) > 0) THEN
				rProductionTime := UDINT_TO_REAL(GoodPieces)* DWORD_TO_REAL(TIME_TO_DWORD(tIdealCycleTime));
				rOperatingTime	:= DWORD_TO_REAL(TIME_TO_DWORD(OperatingTime));
				Performance := rProductionTime / rOperatingTime;			
			ELSE
				Performance := 0;		
			END_IF
			
			OEE := Availabilty * Performance * Quality;
			
			
		IF(TimeStart > EndSessionTime) THEN
			iState := 999;
		END_IF
ELSE
	;
END_CASE

END_PROGRAM

// ---- FCs/FC_Concat4.TcPOU
FUNCTION FC_Concat4 : STRING
VAR_INPUT
    STR1: STRING(255);
    STR2: STRING(255);
    STR3: STRING(255):= '';
    STR4: STRING(255):= '';
    // etc up to a large number
END_VAR
VAR
	
END_VAR



FC_Concat4 := CONCAT(STR1 := FC_Concat4, STR2 := STR1);
FC_Concat4 := CONCAT(STR1 := FC_Concat4, STR2 := STR2);
FC_Concat4 := CONCAT(STR1 := FC_Concat4, STR2 := STR3);
FC_Concat4 := CONCAT(STR1 := FC_Concat4, STR2 := STR4);
// etc up to all defined inputs

END_FUNCTION

// ---- FCs/FC_HeaderCounters.TcPOU
FUNCTION FC_HeaderCounters : UDINT
VAR_INPUT
    In: STRING(50);
	FindLeft : BOOL;
END_VAR
VAR
	tempString	: T_MaxString;
	Pos : INT;
END_VAR

Pos := FIND(In, '/');
IF FindLeft THEN
	tempString := LEFT(In, LEN(In)-Pos);
ELSE
	tempString := RIGHT(In, LEN(In)-Pos);
END_IF

FC_HeaderCounters := STRING_TO_UDINT(tempString);

END_FUNCTION

// ---- FCs/FC_CycleTimeToString.TcPOU
FUNCTION FC_CycleTimeToString : STRING(20);
VAR_INPUT
	CycleTime	: DWORD;
END_VAR
VAR
    TempStr : STRING(20);
    Thousands : UDINT;
    Remainder : UDINT;
	sRemainder : STRING(3);
END_VAR

(* Calcolo delle migliaia e del resto *)
Thousands := CycleTime / 1000;
Remainder := CycleTime MOD 1000;

(* Creazione della stringa con il formato richiesto *)
IF Thousands = 0 THEN
    // Se < 1000: stampiamo il valore diretto
	TempStr := '0.';
    TempStr := CONCAT(TempStr, DWORD_TO_STRING(CycleTime));
ELSE
     // Se >= 1000: separiamo migliaia e resto, es. 10901 -> "10.901"
    TempStr := UDINT_TO_STRING(Thousands);

    // Converto il resto in stringa
    sRemainder := UDINT_TO_STRING(Remainder);

    // Aggiungo eventuali zeri a sinistra, per avere sempre 3 cifre nel resto
    IF LEN(sRemainder) = 1 THEN
        sRemainder := CONCAT('00', sRemainder);
    ELSIF LEN(sRemainder) = 2 THEN
        sRemainder := CONCAT('0', sRemainder);
    END_IF

    // Creo la parte "xxx.yyy"
    TempStr := CONCAT(TempStr, '.');
	TempStr := CONCAT(TempStr, sRemainder);
END_IF;

// Aggiungo la " s" finale
FC_CycleTimeToString := CONCAT(TempStr, ' s');

END_FUNCTION

// ---- FCs/FC_ProductStatus.TcPOU
FUNCTION FC_ProductStatus : eProductStatus
VAR_INPUT
	aByte					: stByteAsBit;
END_VAR

IF aByte.aBit.b0 THEN
	IF aByte.aBit.b1 THEN
		FC_ProductStatus := eProductStatus.Scraped;
	ELSIF aByte.aBit.b3 THEN
		FC_ProductStatus := eProductStatus.Completed;
	ELSIF aByte.aBit.b2 THEN
		FC_ProductStatus := eProductStatus.Working;	
	ELSE
		FC_ProductStatus := eProductStatus.Present;
	END_IF
ELSE
	FC_ProductStatus := eProductStatus.NotPresent;
END_IF

END_FUNCTION

// ---- FBs/Database/PRG_MSSQL_InitConnection.TcPOU
PROGRAM PRG_MSSQL_InitConnection
VAR_INPUT
	Enable			: BOOL;
	DBID			: UDINT;
	tRetryConn		: TIME;
	pSQLCommand1	: POINTER TO FB_SQLCommandEvt;
	pSQLCommand2	: POINTER TO FB_SQLCommandEvt;	
	pSQLCommand3	: POINTER TO FB_SQLCommandEvt;
	pSQLCommand4	: POINTER TO FB_SQLCommandEvt;
	pSQLStoredProcedureEvt	: ARRAY[0..DB.MAX_NUMBER_ST] OF POINTER TO FB_SQLStoredProcedureEvt;
END_VAR
VAR_OUTPUT
	Error			: BOOL;
	ErrorID			: UINT;
	Connected		: BOOL;
END_VAR
VAR
	TON_DelayStartConnection : TON;
	fbSQLDatabaseEvt	: FB_SQLDatabaseEvt(sNetID := '', tTimeout := T#5S);
	fbSqlResult 		: FB_SQLResultEvt(sNetID:='', tTimeout := T#5S);
	iState				: INT := -1;
	RTRIG_Enable		: R_TRIG;
	FTRIG_Enable		: F_TRIG;
	TON_RetryConnection : TON;
	SQLSPParameterSize1		: ARRAY[0..0] OF ST_SQLSPParameter;
	SQLSPParameterSize2		: ARRAY[0..1] OF ST_SQLSPParameter;
	SQLSPParameterSize3		: ARRAY[0..2] OF ST_SQLSPParameter;
	SQLSPParameterSize4		: ARRAY[0..3] OF ST_SQLSPParameter;
	SQLSPParameterSize5		: ARRAY[0..4] OF ST_SQLSPParameter;
	SQLSPParameterSize6		: ARRAY[0..5] OF ST_SQLSPParameter;
END_VAR

RTRIG_Enable(CLK := Enable);
FTRIG_Enable(CLK := Enable);

TON_RetryConnection(IN := iState = 5,PT := tRetryConn);
IF(RTRIG_Enable.Q) THEN
	IF iState = 999 THEN
		iState							:= 2;			// -> Connect	
	ELSE
		iState							:= 0;			// -> Connect	
	END_IF

	
	ErrorID						:= 0;
ELSIF(FTRIG_Enable.Q) THEN	
	
	ErrorID						:= 0;
	iState							:= 990;			// -> Disconnect			
END_IF


TON_DelayStartConnection(IN := iState = 0, PT := T#1m);
CASE iState OF
	-1:
		Connected := FALSE;
		
	0:
		IF TON_DelayStartConnection.Q THEN
			
			iState								:= 2;
		END_IF
		
	 2:
// Connection 
		Connected := FALSE;
		fbSQLDatabaseEvt.Connect(DBID);
		IF(fbSQLDatabaseEvt.bConnected) THEN
			
			iState								:= 10;
		ELSIF(fbSQLDatabaseEvt.bError) THEN
			Error 						:= TRUE;
			ErrorID						:= 1001;
			
			iState								:= 5;
		END_IF
		
	5:	
// Wait time before retry
		IF(TON_RetryConnection.Q) THEN
			ErrorID						:= 0;
			
			iState								:= 2;
		END_IF
		
	10:
		IF(fbSQLDatabaseEvt.CreateCmd(pSQLCommand1)) THEN
			IF(fbSQLDatabaseEvt.bError) THEN
				
				iState							:= 1010;
			ELSE
								

				iState							:= 20;
			END_IF
		END_IF

	20:	
		IF(fbSQLDatabaseEvt.CreateCmd(pSQLCommand2)) THEN
			IF(fbSQLDatabaseEvt.bError) THEN
				
				iState							:= 1020;
			ELSE
								
				iState							:= 30;
			END_IF
		END_IF
		
	30:	
		IF(fbSQLDatabaseEvt.CreateCmd(pSQLCommand3)) THEN
			IF(fbSQLDatabaseEvt.bError) THEN
				
				iState							:= 1030;
			ELSE
								
				iState							:= 40;
			END_IF
		END_IF
		
	40:	
		IF(fbSQLDatabaseEvt.CreateCmd(pSQLCommand4)) THEN
			IF(fbSQLDatabaseEvt.bError) THEN
				
				iState							:= 1040;
			ELSE
		
				iState							:= 50;
			END_IF
		END_IF
		
	50:
		IF fbSQLDatabaseEvt.CreateSP('[dbo].[GetNextPartDataSet]', 0, 0, pSQLStoredProcedureEvt[0]) THEN	
			IF fbSQLDatabaseEvt.bError THEN
	
				iState							:=1050;
			ELSE
				
				iState							:= 60;
			END_IF
		END_IF

// Get PLC Data		
	60:
		SQLSPParameterSize1[0].sParameterName     := '@Id';
		SQLSPParameterSize1[0].eParameterType     := E_SPParameterType.Input;
		SQLSPParameterSize1[0].eParameterDataType := E_ColumnType.BigInt;
		SQLSPParameterSize1[0].nParameterSize     := 8;
		
		IF fbSQLDatabaseEvt.CreateSP('[dbo].[GetPartPLCDataById]', ADR(SQLSPParameterSize1), SIZEOF(SQLSPParameterSize1), pSQLStoredProcedureEvt[1]) THEN	
			IF fbSQLDatabaseEvt.bError THEN
	
				iState							:=1060;
			ELSE
				
				iState							:= 70;
			END_IF
		END_IF

// Get HMI Data
	70:
		IF fbSQLDatabaseEvt.CreateSP('[dbo].[GetPartHMIDataById]', 0, 0, pSQLStoredProcedureEvt[2]) THEN	
			IF fbSQLDatabaseEvt.bError THEN
	
				iState							:=1070;
			ELSE
				
				iState							:= 80;
			END_IF
		END_IF		
		
// Get Order List
	80:
		IF fbSQLDatabaseEvt.CreateSP('[dbo].[GetOrderInfoList]', 0, 0, pSQLStoredProcedureEvt[3]) THEN	
			IF fbSQLDatabaseEvt.bError THEN
	
				iState							:=1080;
			ELSE
				
				iState							:= 90;
			END_IF
		END_IF

// Append order
	90:
		SQLSPParameterSize3[0].sParameterName := '@return';
		SQLSPParameterSize3[0].eParameterType := E_SPParameterType.ReturnValue;
		SQLSPParameterSize3[0].eParameterDataType := E_ColumnType.Integer;
		SQLSPParameterSize3[0].nParameterSize := SIZEOF(DINT);
	
		SQLSPParameterSize3[1].sParameterName := '@BatchInfoJson';
		SQLSPParameterSize3[1].eParameterType := E_SPParameterType.Input;
		SQLSPParameterSize3[1].eParameterDataType := E_ColumnType.NVarChar;
		SQLSPParameterSize3[1].nParameterSize := SIZEOF(STRING(DB.MAX_STRING_SIZE));
		                  
		SQLSPParameterSize3[2].sParameterName := '@BatchItemsJson';
		SQLSPParameterSize3[2].eParameterType := E_SPParameterType.Input;
		SQLSPParameterSize3[2].eParameterDataType := E_ColumnType.NVarChar;
		SQLSPParameterSize3[2].nParameterSize := SIZEOF(STRING(DB.MAX_STRING_SIZE));
		
		IF fbSQLDatabaseEvt.CreateSP('[dbo].[AppendBatchToProductionQueueFromHMI]', ADR(SQLSPParameterSize3), SIZEOF(SQLSPParameterSize3), pSQLStoredProcedureEvt[4]) THEN	
			IF fbSQLDatabaseEvt.bError THEN
    	
				iState							:=1090;
			ELSE
				
				iState							:= 100;
			END_IF
		END_IF

// Modify quantity of an order	
	100:
		SQLSPParameterSize4[0].sParameterName := '@return';
		SQLSPParameterSize4[0].eParameterType := E_SPParameterType.ReturnValue;
		SQLSPParameterSize4[0].eParameterDataType := E_ColumnType.Integer;
		SQLSPParameterSize4[0].nParameterSize := SIZEOF(DINT);
	                      
		SQLSPParameterSize4[1].sParameterName := '@BatchId';
		SQLSPParameterSize4[1].eParameterType := E_SPParameterType.Input;
		SQLSPParameterSize4[1].eParameterDataType := E_ColumnType.NVarChar;
		SQLSPParameterSize4[1].nParameterSize := SIZEOF(STRING(DB.MAX_STRING_SIZE));
		                  
		SQLSPParameterSize4[2].sParameterName := '@BatchInfoJson';
		SQLSPParameterSize4[2].eParameterType := E_SPParameterType.Input;
		SQLSPParameterSize4[2].eParameterDataType := E_ColumnType.NVarChar;
		SQLSPParameterSize4[2].nParameterSize := SIZEOF(STRING(DB.MAX_STRING_SIZE));
		
		SQLSPParameterSize4[3].sParameterName := '@BatchItemsJson';
		SQLSPParameterSize4[3].eParameterType := E_SPParameterType.Input;
		SQLSPParameterSize4[3].eParameterDataType := E_ColumnType.NVarChar;
		SQLSPParameterSize4[3].nParameterSize := SIZEOF(STRING(DB.MAX_STRING_SIZE));
	
		IF fbSQLDatabaseEvt.CreateSP('[dbo].[UpdateBatchToProductionQueue]', ADR(SQLSPParameterSize4), SIZEOF(SQLSPParameterSize4), pSQLStoredProcedureEvt[5]) THEN	
			IF fbSQLDatabaseEvt.bError THEN
    	
				iState							:=1100;
			ELSE
				
				iState							:= 110;
			END_IF
		END_IF

// Delete an order
	110:
		SQLSPParameterSize2[0].sParameterName := '@return';
		SQLSPParameterSize2[0].eParameterType := E_SPParameterType.ReturnValue;
		SQLSPParameterSize2[0].eParameterDataType := E_ColumnType.Integer;
		SQLSPParameterSize2[0].nParameterSize := SIZEOF(DINT);
	                      
		SQLSPParameterSize2[1].sParameterName := '@BatchId';
		SQLSPParameterSize2[1].eParameterType := E_SPParameterType.Input;
		SQLSPParameterSize2[1].eParameterDataType := E_ColumnType.NVarChar;
		SQLSPParameterSize2[1].nParameterSize := SIZEOF(STRING(50));
		
		IF fbSQLDatabaseEvt.CreateSP('[dbo].[DeleteBatchToProductionQueue]', ADR(SQLSPParameterSize2), SIZEOF(SQLSPParameterSize2), pSQLStoredProcedureEvt[6]) THEN	
			IF fbSQLDatabaseEvt.bError THEN
    	
				iState							:=1110;
			ELSE
				
				iState							:= 120;
			END_IF
		END_IF

	120: 
		// Batch Name X
		SQLSPParameterSize2[0].sParameterName := '@BatchNameToMove';
		SQLSPParameterSize2[0].eParameterType := E_SPParameterType.Input;
		SQLSPParameterSize2[0].eParameterDataType := E_ColumnType.NVarChar;
		SQLSPParameterSize2[0].nParameterSize := SIZEOF(STRING(50));
		
		// Batch Name Y
		SQLSPParameterSize2[1].sParameterName := '@NewPos';
		SQLSPParameterSize2[1].eParameterType := E_SPParameterType.Input;
		SQLSPParameterSize2[1].eParameterDataType := E_ColumnType.BigInt;
		SQLSPParameterSize2[1].nParameterSize := SIZEOF(LINT);
		
		IF fbSQLDatabaseEvt.CreateSP('[dbo].[ChangePositionBatchInProductionQueue]', ADR(SQLSPParameterSize2), SIZEOF(SQLSPParameterSize2), pSQLStoredProcedureEvt[7]) THEN
			IF fbSQLDatabaseEvt.bError THEN
	
				iState							:= 1120;
			ELSE
				
				iState							:= 130;
			END_IF
		END_IF

	130:
		SQLSPParameterSize2[0].sParameterName     := '@return';
		SQLSPParameterSize2[0].eParameterType     := E_SPParameterType.ReturnValue;
		SQLSPParameterSize2[0].eParameterDataType := E_ColumnType.Integer;
		SQLSPParameterSize2[0].nParameterSize     := SIZEOF(DINT);
		                   
		SQLSPParameterSize2[1].sParameterName     := '@PLCData';
		SQLSPParameterSize2[1].eParameterType     := E_SPParameterType.Output;
		SQLSPParameterSize2[1].eParameterDataType := E_ColumnType.NVarChar;
		SQLSPParameterSize2[1].nParameterSize     := SIZEOF(STRING(DB.MAX_STRING_SIZE));
		
		IF fbSQLDatabaseEvt.CreateSP('[dbo].[GetNextPartPLCData]', ADR(SQLSPParameterSize2), SIZEOF(SQLSPParameterSize2), pSQLStoredProcedureEvt[8]) THEN	
			IF fbSQLDatabaseEvt.bError THEN
	
				iState							:=1130;
			ELSE
				
				iState							:= 140;
			END_IF
		END_IF		
		
	140:
		SQLSPParameterSize2[0].sParameterName     := '@return';
		SQLSPParameterSize2[0].eParameterType     := E_SPParameterType.ReturnValue;
		SQLSPParameterSize2[0].eParameterDataType := E_ColumnType.Integer;
		SQLSPParameterSize2[0].nParameterSize     := SIZEOF(DINT);
		
		SQLSPParameterSize2[1].sParameterName     := '@PartLocationsAndProcessingDataJson';
		SQLSPParameterSize2[1].eParameterType     := E_SPParameterType.Input;
		SQLSPParameterSize2[1].eParameterDataType := E_ColumnType.NVarChar;
		SQLSPParameterSize2[1].nParameterSize     := SIZEOF(STRING(DB.MAX_STRING_SIZE));
		
		IF fbSQLDatabaseEvt.CreateSP('[dbo].[UpdatePartLocationsAndProcessingData]', ADR(SQLSPParameterSize2), SIZEOF(SQLSPParameterSize2), pSQLStoredProcedureEvt[9]) THEN	
			IF fbSQLDatabaseEvt.bError THEN
	
				iState							:=1140;
			ELSE
				
				iState							:= 150;
			END_IF
		END_IF	
		
	150:
		SQLSPParameterSize2[0].sParameterName := '@return';
		SQLSPParameterSize2[0].eParameterType := E_SPParameterType.ReturnValue;
		SQLSPParameterSize2[0].eParameterDataType := E_ColumnType.Integer;
		SQLSPParameterSize2[0].nParameterSize := SIZEOF(DINT);
		
		SQLSPParameterSize2[1].sParameterName := '@ProcessingData';
		SQLSPParameterSize2[1].eParameterType := E_SPParameterType.Output;
		SQLSPParameterSize2[1].eParameterDataType := E_ColumnType.NVarChar;
		SQLSPParameterSize2[1].nParameterSize := SIZEOF(STRING(DB.MAX_STRING_SIZE));
		
		IF fbSQLDatabaseEvt.CreateSP('[dbo].[GetProcessingDataForHMI]', ADR(SQLSPParameterSize2), SIZEOF(SQLSPParameterSize2), pSQLStoredProcedureEvt[10]) THEN	
			IF fbSQLDatabaseEvt.bError THEN
	
				iState							:=1150;
			ELSE
				
				iState							:= 160;
			END_IF
		END_IF	
		
	160:
		SQLSPParameterSize1[0].sParameterName := '@ProductName';
		SQLSPParameterSize1[0].eParameterType := E_SPParameterType.Input;
		SQLSPParameterSize1[0].eParameterDataType := E_ColumnType.NVarChar;
		SQLSPParameterSize1[0].nParameterSize := SIZEOF(STRING(50));
		
		IF fbSQLDatabaseEvt.CreateSP('[dbo].[GetResourceOrigin]', ADR(SQLSPParameterSize1), SIZEOF(SQLSPParameterSize1), pSQLStoredProcedureEvt[11]) THEN	
			IF fbSQLDatabaseEvt.bError THEN
	
				iState							:=1160;
			ELSE
				
				iState							:= 170;
			END_IF
		END_IF	
		
	170:
		SQLSPParameterSize2[0].sParameterName := '@return';
		SQLSPParameterSize2[0].eParameterType := E_SPParameterType.ReturnValue;
		SQLSPParameterSize2[0].eParameterDataType := E_ColumnType.Integer;
		SQLSPParameterSize2[0].nParameterSize := SIZEOF(DINT);
		
		SQLSPParameterSize2[1].sParameterName := '@jsonAxis';
		SQLSPParameterSize2[1].eParameterType := E_SPParameterType.Input;
		SQLSPParameterSize2[1].eParameterDataType := E_ColumnType.NVarChar;
		SQLSPParameterSize2[1].nParameterSize := SIZEOF(STRING(DB.MAX_STRING_SIZE));
		
		IF fbSQLDatabaseEvt.CreateSP('[dbo].[ModifyOriginAxisInfoToResourceRepository]', ADR(SQLSPParameterSize2), SIZEOF(SQLSPParameterSize2), pSQLStoredProcedureEvt[12]) THEN	
			IF fbSQLDatabaseEvt.bError THEN
	
				iState							:=1170;
			ELSE
				
				iState							:= 180;
			END_IF
		END_IF	
		
	180:
		// Return
		SQLSPParameterSize3[0].sParameterName := '@return';
		SQLSPParameterSize3[0].eParameterType := E_SPParameterType.ReturnValue;
		SQLSPParameterSize3[0].eParameterDataType := E_ColumnType.Integer;
		SQLSPParameterSize3[0].nParameterSize := SIZEOF(DINT);
		
		// BatchName
		SQLSPParameterSize3[1].sParameterName := '@BatchName';
		SQLSPParameterSize3[1].eParameterType := E_SPParameterType.Input;
		SQLSPParameterSize3[1].eParameterDataType := E_ColumnType.NVarChar;
		SQLSPParameterSize3[1].nParameterSize := SIZEOF(STRING(50));
		
		// NewBatchName
		SQLSPParameterSize3[2].sParameterName := '@NewBatchName';
		SQLSPParameterSize3[2].eParameterType := E_SPParameterType.Input;
		SQLSPParameterSize3[2].eParameterDataType := E_ColumnType.NVarChar;
		SQLSPParameterSize3[2].nParameterSize := SIZEOF(STRING(50));
		
		IF fbSQLDatabaseEvt.CreateSP('[dbo].[DuplicateBatchInProductionQueue]', ADR(SQLSPParameterSize3), SIZEOF(SQLSPParameterSize3), pSQLStoredProcedureEvt[13]) THEN	
			IF fbSQLDatabaseEvt.bError THEN
    	
				iState							:=1180;
			ELSE
				
				iState							:= 190;
			END_IF
		END_IF	
		
	190:
		// Return
		SQLSPParameterSize2[0].sParameterName := '@return';
		SQLSPParameterSize2[0].eParameterType := E_SPParameterType.ReturnValue;
		SQLSPParameterSize2[0].eParameterDataType := E_ColumnType.Integer;
		SQLSPParameterSize2[0].nParameterSize := SIZEOF(DINT);
		
		// ResourceType
		SQLSPParameterSize2[1].sParameterName := '@ResourceType';
		SQLSPParameterSize2[1].eParameterType := E_SPParameterType.Input;
		SQLSPParameterSize2[1].eParameterDataType := E_ColumnType.NVarChar;
		SQLSPParameterSize2[1].nParameterSize := SIZEOF(STRING(50));
		
		IF fbSQLDatabaseEvt.CreateSP('[dbo].[GetResourcesByType]', ADR(SQLSPParameterSize2), SIZEOF(SQLSPParameterSize2), pSQLStoredProcedureEvt[14]) THEN	
			IF fbSQLDatabaseEvt.bError THEN
    	
				iState							:=1190;
			ELSE
				
				iState							:= 200;
			END_IF
		END_IF	
		
	200:
		// Return
		SQLSPParameterSize2[0].sParameterName := '@return';
		SQLSPParameterSize2[0].eParameterType := E_SPParameterType.ReturnValue;
		SQLSPParameterSize2[0].eParameterDataType := E_ColumnType.Integer;
		SQLSPParameterSize2[0].nParameterSize := SIZEOF(DINT);
		
		// ResourceName
		SQLSPParameterSize2[1].sParameterName := '@ResourceName';
		SQLSPParameterSize2[1].eParameterType := E_SPParameterType.Input;
		SQLSPParameterSize2[1].eParameterDataType := E_ColumnType.NVarChar;
		SQLSPParameterSize2[1].nParameterSize := SIZEOF(STRING(50));
		IF fbSQLDatabaseEvt.CreateSP('[dbo].[GetResourcesByName]', ADR(SQLSPParameterSize2), SIZEOF(SQLSPParameterSize2), pSQLStoredProcedureEvt[15]) THEN	
			IF fbSQLDatabaseEvt.bError THEN
    	
				iState							:=1200;
			ELSE
				
				iState							:= 210;
			END_IF
		END_IF	
		
	210:
		// Return
		SQLSPParameterSize3[0].sParameterName := '@return';
		SQLSPParameterSize3[0].eParameterType := E_SPParameterType.ReturnValue;
		SQLSPParameterSize3[0].eParameterDataType := E_ColumnType.Integer;
		SQLSPParameterSize3[0].nParameterSize := SIZEOF(DINT);
		
		// ResourceName
		SQLSPParameterSize3[1].sParameterName := '@ResourceName';
		SQLSPParameterSize3[1].eParameterType := E_SPParameterType.Input;
		SQLSPParameterSize3[1].eParameterDataType := E_ColumnType.NVarChar;
		SQLSPParameterSize3[1].nParameterSize := SIZEOF(STRING(50));
		
		// ResourceName
		SQLSPParameterSize3[2].sParameterName := '@NewData';
		SQLSPParameterSize3[2].eParameterType := E_SPParameterType.Input;
		SQLSPParameterSize3[2].eParameterDataType := E_ColumnType.NVarChar;
		SQLSPParameterSize3[2].nParameterSize := SIZEOF(STRING(DB.MAX_STRING_SIZE));
		
		IF fbSQLDatabaseEvt.CreateSP('[dbo].[SetResourcesByName]', ADR(SQLSPParameterSize3), SIZEOF(SQLSPParameterSize3), pSQLStoredProcedureEvt[16]) THEN	
			IF fbSQLDatabaseEvt.bError THEN
    	
				iState							:=1210;
			ELSE
				
				iState							:= 220;
			END_IF
		END_IF	
		
	220:
		// Return
		SQLSPParameterSize2[0].sParameterName := '@return';
		SQLSPParameterSize2[0].eParameterType := E_SPParameterType.ReturnValue;
		SQLSPParameterSize2[0].eParameterDataType := E_ColumnType.Integer;
		SQLSPParameterSize2[0].nParameterSize := SIZEOF(DINT);
		
		// ResourceType
		SQLSPParameterSize2[1].sParameterName := '@ResourceType';
		SQLSPParameterSize2[1].eParameterType := E_SPParameterType.Input;
		SQLSPParameterSize2[1].eParameterDataType := E_ColumnType.NVarChar;
		SQLSPParameterSize2[1].nParameterSize := SIZEOF(STRING(50));
		
		IF fbSQLDatabaseEvt.CreateSP('[dbo].[GetResourcesListByType]', ADR(SQLSPParameterSize2), SIZEOF(SQLSPParameterSize2), pSQLStoredProcedureEvt[17]) THEN	
			IF fbSQLDatabaseEvt.bError THEN
    	
				iState							:=1220;
			ELSE
				
				iState							:= 230;
			END_IF
		END_IF	
		
	230:
		// Return
		SQLSPParameterSize2[0].sParameterName := '@return';
		SQLSPParameterSize2[0].eParameterType := E_SPParameterType.ReturnValue;
		SQLSPParameterSize2[0].eParameterDataType := E_ColumnType.Integer;
		SQLSPParameterSize2[0].nParameterSize := SIZEOF(DINT);
		
		// ResourceType
		SQLSPParameterSize2[1].sParameterName := '@SequenceName';
		SQLSPParameterSize2[1].eParameterType := E_SPParameterType.Input;
		SQLSPParameterSize2[1].eParameterDataType := E_ColumnType.NVarChar;
		SQLSPParameterSize2[1].nParameterSize := SIZEOF(STRING(50));
		
		IF fbSQLDatabaseEvt.CreateSP('[dbo].[GetFormattedTablesFromSequences]', ADR(SQLSPParameterSize2), SIZEOF(SQLSPParameterSize2), pSQLStoredProcedureEvt[18]) THEN	
			IF fbSQLDatabaseEvt.bError THEN
    	
				iState							:=1230;
			ELSE
				
				iState							:= 240;
			END_IF
		END_IF	
		
	240:
		// Return
		SQLSPParameterSize2[0].sParameterName := '@return';
		SQLSPParameterSize2[0].eParameterType := E_SPParameterType.ReturnValue;
		SQLSPParameterSize2[0].eParameterDataType := E_ColumnType.Integer;
		SQLSPParameterSize2[0].nParameterSize := SIZEOF(DINT);
		
		// ResourceType
		SQLSPParameterSize2[1].sParameterName := '@SequenceName';
		SQLSPParameterSize2[1].eParameterType := E_SPParameterType.Input;
		SQLSPParameterSize2[1].eParameterDataType := E_ColumnType.NVarChar;
		SQLSPParameterSize2[1].nParameterSize := SIZEOF(STRING(50));
		
		IF fbSQLDatabaseEvt.CreateSP('[dbo].[GetOriginsFromSequence]', ADR(SQLSPParameterSize2), SIZEOF(SQLSPParameterSize2), pSQLStoredProcedureEvt[19]) THEN	
			IF fbSQLDatabaseEvt.bError THEN
    	
				iState							:=1240;
			ELSE
				
				iState							:= 250;
			END_IF
		END_IF	
		
	250:
		IF fbSQLDatabaseEvt.CreateSP('[dbo].[GetOrigins]', 0, 0, pSQLStoredProcedureEvt[20]) THEN	
			IF fbSQLDatabaseEvt.bError THEN
    	
				iState							:=1250;
			ELSE
				
				iState							:= 260;
			END_IF
		END_IF	

	260:
		SQLSPParameterSize1[0].sParameterName := '@Name';
		SQLSPParameterSize1[0].eParameterType := E_SPParameterType.Input;
		SQLSPParameterSize1[0].eParameterDataType := E_ColumnType.NVarChar;
		SQLSPParameterSize1[0].nParameterSize := SIZEOF(STRING(50));
		
		IF fbSQLDatabaseEvt.CreateSP('[dbo].[GetOriginsByName]', ADR(SQLSPParameterSize1), SIZEOF(SQLSPParameterSize1), pSQLStoredProcedureEvt[21]) THEN	
			IF fbSQLDatabaseEvt.bError THEN
    	
				iState							:=1260;
			ELSE
				
				iState							:= 270;
			END_IF
		END_IF
		
	270:
		SQLSPParameterSize1[0].sParameterName := '@Size';
		SQLSPParameterSize1[0].eParameterType := E_SPParameterType.Input;
		SQLSPParameterSize1[0].eParameterDataType := E_ColumnType.Integer;
		SQLSPParameterSize1[0].nParameterSize := SIZEOF(DINT);
		
		IF fbSQLDatabaseEvt.CreateSP('[dbo].[GetOriginsBySide]', ADR(SQLSPParameterSize1), SIZEOF(SQLSPParameterSize1), pSQLStoredProcedureEvt[22]) THEN	
			IF fbSQLDatabaseEvt.bError THEN
    	
				iState							:=1270;
			ELSE
				
				iState							:= 280;
			END_IF
		END_IF
		
	280:
		IF fbSQLDatabaseEvt.CreateSP('[dbo].[GetCutters]', 0, 0, pSQLStoredProcedureEvt[23]) THEN	
			IF fbSQLDatabaseEvt.bError THEN
    	
				iState							:=1280;
			ELSE
				
				iState							:= 290;
			END_IF
		END_IF	

	290:
		SQLSPParameterSize1[0].sParameterName := '@Name';
		SQLSPParameterSize1[0].eParameterType := E_SPParameterType.Input;
		SQLSPParameterSize1[0].eParameterDataType := E_ColumnType.NVarChar;
		SQLSPParameterSize1[0].nParameterSize := SIZEOF(STRING(50));
		
		IF fbSQLDatabaseEvt.CreateSP('[dbo].[GetCuttersByName]', ADR(SQLSPParameterSize1), SIZEOF(SQLSPParameterSize1), pSQLStoredProcedureEvt[24]) THEN	
			IF fbSQLDatabaseEvt.bError THEN
    	
				iState							:=1290;
			ELSE
				
				iState							:= 300;
			END_IF
		END_IF
		
	300:
		SQLSPParameterSize1[0].sParameterName := '@Size';
		SQLSPParameterSize1[0].eParameterType := E_SPParameterType.Input;
		SQLSPParameterSize1[0].eParameterDataType := E_ColumnType.Integer;
		SQLSPParameterSize1[0].nParameterSize := SIZEOF(DINT);
		
		IF fbSQLDatabaseEvt.CreateSP('[dbo].[GetCuttersBySide]', ADR(SQLSPParameterSize1), SIZEOF(SQLSPParameterSize1), pSQLStoredProcedureEvt[25]) THEN	
			IF fbSQLDatabaseEvt.bError THEN
    	
				iState							:=1300;
			ELSE
				
				iState							:= 310;
			END_IF
		END_IF
		
	310:
		IF fbSQLDatabaseEvt.CreateSP('[dbo].[GetMillings]', 0, 0, pSQLStoredProcedureEvt[26]) THEN	
			IF fbSQLDatabaseEvt.bError THEN
    	
				iState							:=1310;
			ELSE
				
				iState							:= 320;
			END_IF
		END_IF	

	320:
		SQLSPParameterSize1[0].sParameterName := '@Name';
		SQLSPParameterSize1[0].eParameterType := E_SPParameterType.Input;
		SQLSPParameterSize1[0].eParameterDataType := E_ColumnType.NVarChar;
		SQLSPParameterSize1[0].nParameterSize := SIZEOF(STRING(50));
		
		IF fbSQLDatabaseEvt.CreateSP('[dbo].[GetMillingsByName]', ADR(SQLSPParameterSize1), SIZEOF(SQLSPParameterSize1), pSQLStoredProcedureEvt[27]) THEN	
			IF fbSQLDatabaseEvt.bError THEN
    	
				iState							:=1320;
			ELSE
				
				iState							:= 330;
			END_IF
		END_IF
		
	330:
		SQLSPParameterSize1[0].sParameterName := '@FamilyName';
		SQLSPParameterSize1[0].eParameterType := E_SPParameterType.Input;
		SQLSPParameterSize1[0].eParameterDataType := E_ColumnType.NVarChar;
		SQLSPParameterSize1[0].nParameterSize := SIZEOF(STRING(50));
		
		IF fbSQLDatabaseEvt.CreateSP('[dbo].[GetMillingsByFamilyName]', ADR(SQLSPParameterSize1), SIZEOF(SQLSPParameterSize1), pSQLStoredProcedureEvt[28]) THEN	
			IF fbSQLDatabaseEvt.bError THEN
    	
				iState							:=1330;
			ELSE
				
				iState							:= 340;
			END_IF
		END_IF
		
	340:
		SQLSPParameterSize1[0].sParameterName := '@GetResourcesByNameMilling';
		SQLSPParameterSize1[0].eParameterType := E_SPParameterType.Input;
		SQLSPParameterSize1[0].eParameterDataType := E_ColumnType.NVarChar;
		SQLSPParameterSize1[0].nParameterSize := SIZEOF(STRING(50));
		
